  [680] = {x=34.462, y=0.000, z=-5.329, rx=-0.000, ry=0.000, rz=-0.000, shoulder=lefty, elbow=epositive, wrist=wpositive, fatherId=fReference[0]}
  [681] = {x=33.526, y=0.000, z=-5.347, rx=-0.000, ry=0.000, rz=-0.000, shoulder=lefty, elbow=epositive, wrist=wpositive, fatherId=fReference[0]}
  [682] = {x=32.941, y=0.000, z=-5.345, rx=-0.000, ry=0.000, rz=-0.000, shoulder=lefty, elbow=epositive, wrist=wpositive, fatherId=fReference[0]}
  [683] = {x=32.394, y=0.000, z=-5.347, rx=-0.000, ry=0.000, rz=-0.000, shoulder=lefty, elbow=epositive, wrist=wpositive, fatherId=fReference[0]}
  [684] = {x=31.868, y=0.000, z=-5.351, rx=-0.000, ry=0.000, rz=-0.000, shoulder=lefty, elbow=epositive, wrist=wpositive, fatherId=fReference[0]}
  [685] = {x=31.351, y=0.000, z=-5.356, rx=-0.000, ry=0.000, rz=-0.000, shoulder=lefty, elbow=epositive, wrist=wpositive, fatherId=fReference[0]}
  [686] = {x=30.840, y=0.000, z=-5.362, rx=-0.000, ry=0.000, rz=-0.000, shoulder=lefty, elbow=epositive, wrist=wpositive, fatherId=fReference[0]}
  [687] = {x=30.332, y=0.000, z=-5.369, rx=-0.000, ry=0.000, rz=-0.000, shoulder=lefty, elbow=epositive, wrist=wpositive, fatherId=fReference[0]}
  [688] = {x=29.826, y=0.000, z=-5.375, rx=-0.000, ry=0.000, rz=-0.000, shoulder=lefty, elbow=epositive, wrist=wpositive, fatherId=fReference[0]}
  [689] = {x=29.322, y=0.000, z=-5.383, rx=-0.000, ry=0.000, rz=-0.000, shoulder=lefty, elbow=epositive, wrist=wpositive, fatherId=fReference[0]}
  [690] = {x=28.818, y=0.000, z=-5.390, rx=-0.000, ry=0.000, rz=-0.000, shoulder=lefty, elbow=epositive, wrist=wpositive, fatherId=fReference[0]}
  [691] = {x=28.316, y=0.000, z=-5.397, rx=-0.000, ry=0.000, rz=-0.000, shoulder=lefty, elbow=epositive, wrist=wpositive, fatherId=fReference[0]}
  [692] = {x=27.814, y=0.000, z=-5.405, rx=-0.000, ry=0.000, rz=-0.000, shoulder=lefty, elbow=epositive, wrist=wpositive, fatherId=fReference[0]}
  [693] = {x=27.312, y=0.000, z=-5.413, rx=-0.000, ry=0.000, rz=-0.000, shoulder=lefty, elbow=epositive, wrist=wpositive, fatherId=fReference[0]}
  [694] = {x=26.812, y=0.000, z=-5.421, rx=-0.000, ry=0.000, rz=-0.000, shoulder=lefty, elbow=epositive, wrist=wpositive, fatherId=fReference[0]}
  [695] = {x=26.312, y=0.000, z=-5.429, rx=-0.000, ry=0.000, rz=-0.000, shoulder=lefty, elbow=epositive, wrist=wpositive, fatherId=fReference[0]}
  [696] = {x=25.812, y=0.000, z=-5.437, rx=-0.000, ry=0.000, rz=-0.000, shoulder=lefty, elbow=epositive, wrist=wpositive, fatherId=fReference[0]}
  [697] = {x=25.313, y=0.000, z=-5.446, rx=-0.000, ry=0.000, rz=-0.000, shoulder=lefty, elbow=epositive, wrist=wpositive, fatherId=fReference[0]}
  [698] = {x=24.813, y=0.000, z=-5.454, rx=-0.000, ry=0.000, rz=-0.000, shoulder=lefty, elbow=epositive, wrist=wpositive, fatherId=fReference[0]}
  [699] = {x=24.314, y=0.000, z=-5.462, rx=-0.000, ry=0.000, rz=-0.000, shoulder=lefty, elbow=epositive, wrist=wpositive, fatherId=fReference[0]}
  [700] = {x=23.815, y=0.000, z=-5.471, rx=-0.000, ry=0.000, rz=-0.000, shoulder=lefty, elbow=epositive, wrist=wpositive, fatherId=fReference[0]}
  [701] = {x=23.315, y=0.000, z=-5.479, rx=-0.000, ry=0.000, rz=-0.000, shoulder=lefty, elbow=epositive, wrist=wpositive, fatherId=fReference[0]}
  [702] = {x=22.816, y=0.000, z=-5.487, rx=-0.000, ry=0.000, rz=-0.000, shoulder=lefty, elbow=epositive, wrist=wpositive, fatherId=fReference[0]}
  [703] = {x=22.317, y=0.000, z=-5.496, rx=-0.000, ry=0.000, rz=-0.000, shoulder=lefty, elbow=epositive, wrist=wpositive, fatherId=fReference[0]}
  [704] = {x=21.818, y=0.000, z=-5.504, rx=-0.000, ry=0.000, rz=-0.000, shoulder=lefty, elbow=epositive, wrist=wpositive, fatherId=fReference[0]}
  [705] = {x=21.319, y=0.000, z=-5.513, rx=-0.000, ry=0.000, rz=-0.000, shoulder=lefty, elbow=epositive, wrist=wpositive, fatherId=fReference[0]}
  [706] = {x=20.820, y=0.000, z=-5.521, rx=-0.000, ry=0.000, rz=-0.000, shoulder=lefty, elbow=epositive, wrist=wpositive, fatherId=fReference[0]}
  [707] = {x=20.321, y=0.000, z=-5.530, rx=-0.000, ry=0.000, rz=-0.000, shoulder=lefty, elbow=epositive, wrist=wpositive, fatherId=fReference[0]}
  [708] = {x=19.823, y=0.000, z=-5.539, rx=-0.000, ry=0.000, rz=-0.000, shoulder=lefty, elbow=epositive, wrist=wpositive, fatherId=fReference[0]}
  [709] = {x=19.325, y=0.000, z=-5.548, rx=-0.000, ry=0.000, rz=-0.000, shoulder=lefty, elbow=epositive, wrist=wpositive, fatherId=fReference[0]}
  [710] = {x=18.827, y=0.000, z=-5.557, rx=-0.000, ry=0.000, rz=-0.000, shoulder=lefty, elbow=epositive, wrist=wpositive, fatherId=fReference[0]}
  [711] = {x=18.328, y=0.000, z=-5.565, rx=-0.000, ry=0.000, rz=-0.000, shoulder=lefty, elbow=epositive, wrist=wpositive, fatherId=fReference[0]}
  [712] = {x=17.830, y=0.000, z=-5.575, rx=-0.000, ry=0.000, rz=-0.000, shoulder=lefty, elbow=epositive, wrist=wpositive, fatherId=fReference[0]}
  [713] = {x=17.331, y=0.000, z=-5.583, rx=-0.000, ry=0.000, rz=-0.000, shoulder=lefty, elbow=epositive, wrist=wpositive, fatherId=fReference[0]}
  [714] = {x=16.833, y=0.000, z=-5.593, rx=-0.000, ry=0.000, rz=-0.000, shoulder=lefty, elbow=epositive, wrist=wpositive, fatherId=fReference[0]}
  [715] = {x=16.335, y=0.000, z=-5.601, rx=-0.000, ry=0.000, rz=-0.000, shoulder=lefty, elbow=epositive, wrist=wpositive, fatherId=fReference[0]}
  [716] = {x=15.836, y=0.000, z=-5.611, rx=-0.000, ry=0.000, rz=-0.000, shoulder=lefty, elbow=epositive, wrist=wpositive, fatherId=fReference[0]}
  [717] = {x=15.338, y=0.000, z=-5.620, rx=-0.000, ry=0.000, rz=-0.000, shoulder=lefty, elbow=epositive, wrist=wpositive, fatherId=fReference[0]}
  [718] = {x=14.840, y=0.000, z=-5.628, rx=-0.000, ry=0.000, rz=-0.000, shoulder=lefty, elbow=epositive, wrist=wpositive, fatherId=fReference[0]}
  [719] = {x=14.342, y=0.000, z=-5.638, rx=-0.000, ry=0.000, rz=-0.000, shoulder=lefty, elbow=epositive, wrist=wpositive, fatherId=fReference[0]}
  [720] = {x=13.843, y=0.000, z=-5.646, rx=-0.000, ry=0.000, rz=-0.000, shoulder=lefty, elbow=epositive, wrist=wpositive, fatherId=fReference[0]}
  [721] = {x=13.344, y=0.000, z=-5.655, rx=-0.000, ry=0.000, rz=-0.000, shoulder=lefty, elbow=epositive, wrist=wpositive, fatherId=fReference[0]}
  [722] = {x=12.846, y=0.000, z=-5.664, rx=-0.000, ry=0.000, rz=-0.000, shoulder=lefty, elbow=epositive, wrist=wpositive, fatherId=fReference[0]}
  [723] = {x=12.345, y=0.000, z=-5.673, rx=-0.000, ry=0.000, rz=-0.000, shoulder=lefty, elbow=epositive, wrist=wpositive, fatherId=fReference[0]}
  [724] = {x=11.846, y=0.000, z=-5.682, rx=-0.000, ry=0.000, rz=-0.000, shoulder=lefty, elbow=epositive, wrist=wpositive, fatherId=fReference[0]}
  [725] = {x=11.347, y=0.000, z=-5.690, rx=-0.000, ry=0.000, rz=-0.000, shoulder=lefty, elbow=epositive, wrist=wpositive, fatherId=fReference[0]}
  [726] = {x=10.847, y=0.000, z=-5.699, rx=-0.000, ry=0.000, rz=-0.000, shoulder=lefty, elbow=epositive, wrist=wpositive, fatherId=fReference[0]}
  [727] = {x=10.347, y=0.000, z=-5.707, rx=-0.000, ry=0.000, rz=-0.000, shoulder=lefty, elbow=epositive, wrist=wpositive, fatherId=fReference[0]}
  [728] = {x=9.846, y=0.000, z=-5.716, rx=-0.000, ry=0.000, rz=-0.000, shoulder=lefty, elbow=epositive, wrist=wpositive, fatherId=fReference[0]}
  [729] = {x=9.346, y=0.000, z=-5.724, rx=-0.000, ry=0.000, rz=-0.000, shoulder=lefty, elbow=epositive, wrist=wpositive, fatherId=fReference[0]}
  [730] = {x=8.847, y=0.000, z=-5.733, rx=-0.000, ry=0.000, rz=-0.000, shoulder=lefty, elbow=epositive, wrist=wpositive, fatherId=fReference[0]}
  [731] = {x=8.346, y=0.000, z=-5.741, rx=-0.000, ry=0.000, rz=-0.000, shoulder=lefty, elbow=epositive, wrist=wpositive, fatherId=fReference[0]}
  [732] = {x=7.846, y=0.000, z=-5.750, rx=-0.000, ry=0.000, rz=-0.000, shoulder=lefty, elbow=epositive, wrist=wpositive, fatherId=fReference[0]}
  [733] = {x=7.344, y=0.000, z=-5.758, rx=-0.000, ry=0.000, rz=-0.000, shoulder=lefty, elbow=epositive, wrist=wpositive, fatherId=fReference[0]}
  [734] = {x=6.843, y=0.000, z=-5.766, rx=-0.000, ry=0.000, rz=-0.000, shoulder=lefty, elbow=epositive, wrist=wpositive, fatherId=fReference[0]}
  [735] = {x=6.341, y=0.000, z=-5.774, rx=-0.000, ry=0.000, rz=-0.000, shoulder=lefty, elbow=epositive, wrist=wpositive, fatherId=fReference[0]}
  [736] = {x=5.838, y=0.000, z=-5.782, rx=-0.000, ry=0.000, rz=-0.000, shoulder=lefty, elbow=epositive, wrist=wpositive, fatherId=fReference[0]}
  [737] = {x=5.336, y=0.000, z=-5.791, rx=-0.000, ry=0.000, rz=-0.000, shoulder=lefty, elbow=epositive, wrist=wpositive, fatherId=fReference[0]}
  [738] = {x=4.831, y=0.000, z=-5.798, rx=-0.000, ry=0.000, rz=-0.000, shoulder=lefty, elbow=epositive, wrist=wpositive, fatherId=fReference[0]}
  [739] = {x=4.326, y=0.000, z=-5.806, rx=-0.000, ry=0.000, rz=-0.000, shoulder=lefty, elbow=epositive, wrist=wpositive, fatherId=fReference[0]}
  [740] = {x=3.823, y=0.000, z=-5.814, rx=-0.000, ry=0.000, rz=-0.000, shoulder=lefty, elbow=epositive, wrist=wpositive, fatherId=fReference[0]}
  [741] = {x=3.321, y=0.000, z=-5.822, rx=-0.000, ry=0.000, rz=-0.000, shoulder=lefty, elbow=epositive, wrist=wpositive, fatherId=fReference[0]}
  [742] = {x=2.818, y=0.000, z=-5.830, rx=-0.000, ry=0.000, rz=-0.000, shoulder=lefty, elbow=epositive, wrist=wpositive, fatherId=fReference[0]}
  [743] = {x=2.316, y=0.000, z=-5.838, rx=-0.000, ry=0.000, rz=-0.000, shoulder=lefty, elbow=epositive, wrist=wpositive, fatherId=fReference[0]}
  [744] = {x=1.816, y=0.000, z=-5.847, rx=-0.000, ry=0.000, rz=-0.000, shoulder=lefty, elbow=epositive, wrist=wpositive, fatherId=fReference[0]}
  [745] = {x=1.313, y=0.000, z=-5.855, rx=-0.000, ry=0.000, rz=-0.000, shoulder=lefty, elbow=epositive, wrist=wpositive, fatherId=fReference[0]}
  [746] = {x=0.814, y=0.000, z=-5.864, rx=-0.000, ry=0.000, rz=-0.000, shoulder=lefty, elbow=epositive, wrist=wpositive, fatherId=fReference[0]}
  [747] = {x=0.312, y=0.000, z=-5.872, rx=-0.000, ry=0.000, rz=-0.000, shoulder=lefty, elbow=epositive, wrist=wpositive, fatherId=fReference[0]}
  [748] = {x=-0.190, y=0.000, z=-5.880, rx=-0.000, ry=0.000, rz=-0.000, shoulder=lefty, elbow=epositive, wrist=wpositive, fatherId=fReference[0]}
  [749] = {x=-0.691, y=0.000, z=-5.889, rx=-0.000, ry=0.000, rz=-0.000, shoulder=lefty, elbow=epositive, wrist=wpositive, fatherId=fReference[0]}
  [750] = {x=-1.192, y=0.000, z=-5.897, rx=-0.000, ry=0.000, rz=-0.000, shoulder=lefty, elbow=epositive, wrist=wpositive, fatherId=fReference[0]}
  [751] = {x=-1.693, y=0.000, z=-5.906, rx=-0.000, ry=0.000, rz=-0.000, shoulder=lefty, elbow=epositive, wrist=wpositive, fatherId=fReference[0]}
  [752] = {x=-2.194, y=0.000, z=-5.915, rx=-0.000, ry=0.000, rz=-0.000, shoulder=lefty, elbow=epositive, wrist=wpositive, fatherId=fReference[0]}
  [753] = {x=-2.695, y=0.000, z=-5.923, rx=-0.000, ry=0.000, rz=-0.000, shoulder=lefty, elbow=epositive, wrist=wpositive, fatherId=fReference[0]}
  [754] = {x=-3.197, y=0.000, z=-5.932, rx=-0.000, ry=0.000, rz=-0.000, shoulder=lefty, elbow=epositive, wrist=wpositive, fatherId=fReference[0]}
  [755] = {x=-3.697, y=0.000, z=-5.941, rx=-0.000, ry=0.000, rz=-0.000, shoulder=lefty, elbow=epositive, wrist=wpositive, fatherId=fReference[0]}
  [756] = {x=-4.197, y=0.000, z=-5.950, rx=-0.000, ry=0.000, rz=-0.000, shoulder=lefty, elbow=epositive, wrist=wpositive, fatherId=fReference[0]}
  [757] = {x=-4.697, y=0.000, z=-5.959, rx=-0.000, ry=0.000, rz=-0.000, shoulder=lefty, elbow=epositive, wrist=wpositive, fatherId=fReference[0]}
  [758] = {x=-5.197, y=0.000, z=-5.968, rx=-0.000, ry=0.000, rz=-0.000, shoulder=lefty, elbow=epositive, wrist=wpositive, fatherId=fReference[0]}
  [759] = {x=-5.696, y=0.000, z=-5.977, rx=-0.000, ry=0.000, rz=-0.000, shoulder=lefty, elbow=epositive, wrist=wpositive, fatherId=fReference[0]}
  [760] = {x=-6.198, y=0.000, z=-5.985, rx=-0.000, ry=0.000, rz=-0.000, shoulder=lefty, elbow=epositive, wrist=wpositive, fatherId=fReference[0]}
  [761] = {x=-6.700, y=0.000, z=-5.994, rx=-0.000, ry=0.000, rz=-0.000, shoulder=lefty, elbow=epositive, wrist=wpositive, fatherId=fReference[0]}
  [762] = {x=-7.198, y=0.000, z=-6.004, rx=-0.000, ry=0.000, rz=-0.000, shoulder=lefty, elbow=epositive, wrist=wpositive, fatherId=fReference[0]}
  [763] = {x=-7.696, y=0.000, z=-6.013, rx=-0.000, ry=0.000, rz=-0.000, shoulder=lefty, elbow=epositive, wrist=wpositive, fatherId=fReference[0]}
  [764] = {x=-8.197, y=0.000, z=-6.022, rx=-0.000, ry=0.000, rz=-0.000, shoulder=lefty, elbow=epositive, wrist=wpositive, fatherId=fReference[0]}
  [765] = {x=-8.698, y=0.000, z=-6.031, rx=-0.000, ry=0.000, rz=-0.000, shoulder=lefty, elbow=epositive, wrist=wpositive, fatherId=fReference[0]}
  [766] = {x=-9.196, y=0.000, z=-6.040, rx=-0.000, ry=0.000, rz=-0.000, shoulder=lefty, elbow=epositive, wrist=wpositive, fatherId=fReference[0]}
  [767] = {x=-9.696, y=0.000, z=-6.050, rx=-0.000, ry=0.000, rz=-0.000, shoulder=lefty, elbow=epositive, wrist=wpositive, fatherId=fReference[0]}
  [768] = {x=-10.193, y=0.000, z=-6.060, rx=-0.000, ry=0.000, rz=-0.000, shoulder=lefty, elbow=epositive, wrist=wpositive, fatherId=fReference[0]}
  [769] = {x=-10.692, y=0.000, z=-6.069, rx=-0.000, ry=0.000, rz=-0.000, shoulder=lefty, elbow=epositive, wrist=wpositive, fatherId=fReference[0]}
  [770] = {x=-11.189, y=0.000, z=-6.079, rx=-0.000, ry=0.000, rz=-0.000, shoulder=lefty, elbow=epositive, wrist=wpositive, fatherId=fReference[0]}
  [771] = {x=-11.687, y=0.000, z=-6.088, rx=-0.000, ry=0.000, rz=-0.000, shoulder=lefty, elbow=epositive, wrist=wpositive, fatherId=fReference[0]}
  [772] = {x=-12.183, y=0.000, z=-6.098, rx=-0.000, ry=0.000, rz=-0.000, shoulder=lefty, elbow=epositive, wrist=wpositive, fatherId=fReference[0]}
  [773] = {x=-12.685, y=0.000, z=-6.108, rx=-0.000, ry=0.000, rz=-0.000, shoulder=lefty, elbow=epositive, wrist=wpositive, fatherId=fReference[0]}
  [774] = {x=-13.181, y=0.000, z=-6.117, rx=-0.000, ry=0.000, rz=-0.000, shoulder=lefty, elbow=epositive, wrist=wpositive, fatherId=fReference[0]}
  [775] = {x=-13.678, y=0.000, z=-6.127, rx=-0.000, ry=0.000, rz=-0.000, shoulder=lefty, elbow=epositive, wrist=wpositive, fatherId=fReference[0]}
  [776] = {x=-14.176, y=0.000, z=-6.137, rx=-0.000, ry=0.000, rz=-0.000, shoulder=lefty, elbow=epositive, wrist=wpositive, fatherId=fReference[0]}
  [777] = {x=-14.670, y=0.000, z=-6.147, rx=-0.000, ry=0.000, rz=-0.000, shoulder=lefty, elbow=epositive, wrist=wpositive, fatherId=fReference[0]}
  [778] = {x=-15.170, y=0.000, z=-6.157, rx=-0.000, ry=0.000, rz=-0.000, shoulder=lefty, elbow=epositive, wrist=wpositive, fatherId=fReference[0]}
  [779] = {x=-15.665, y=0.000, z=-6.167, rx=-0.000, ry=0.000, rz=-0.000, shoulder=lefty, elbow=epositive, wrist=wpositive, fatherId=fReference[0]}
  [780] = {x=-16.162, y=0.000, z=-6.177, rx=-0.000, ry=0.000, rz=-0.000, shoulder=lefty, elbow=epositive, wrist=wpositive, fatherId=fReference[0]}
  [781] = {x=-16.658, y=0.000, z=-6.188, rx=-0.000, ry=0.000, rz=-0.000, shoulder=lefty, elbow=epositive, wrist=wpositive, fatherId=fReference[0]}
  [782] = {x=-17.157, y=0.000, z=-6.197, rx=-0.000, ry=0.000, rz=-0.000, shoulder=lefty, elbow=epositive, wrist=wpositive, fatherId=fReference[0]}
  [783] = {x=-17.653, y=0.000, z=-6.207, rx=-0.000, ry=0.000, rz=-0.000, shoulder=lefty, elbow=epositive, wrist=wpositive, fatherId=fReference[0]}
  [784] = {x=-18.149, y=0.000, z=-6.218, rx=-0.000, ry=0.000, rz=-0.000, shoulder=lefty, elbow=epositive, wrist=wpositive, fatherId=fReference[0]}
  [785] = {x=-18.646, y=0.000, z=-6.228, rx=-0.000, ry=0.000, rz=-0.000, shoulder=lefty, elbow=epositive, wrist=wpositive, fatherId=fReference[0]}
  [786] = {x=-19.137, y=0.000, z=-6.239, rx=-0.000, ry=0.000, rz=-0.000, shoulder=lefty, elbow=epositive, wrist=wpositive, fatherId=fReference[0]}
  [787] = {x=-19.637, y=0.000, z=-6.248, rx=-0.000, ry=0.000, rz=-0.000, shoulder=lefty, elbow=epositive, wrist=wpositive, fatherId=fReference[0]}
  [788] = {x=-20.133, y=0.000, z=-6.259, rx=-0.000, ry=0.000, rz=-0.000, shoulder=lefty, elbow=epositive, wrist=wpositive, fatherId=fReference[0]}
  [789] = {x=-20.628, y=0.000, z=-6.269, rx=-0.000, ry=0.000, rz=-0.000, shoulder=lefty, elbow=epositive, wrist=wpositive, fatherId=fReference[0]}
  [790] = {x=-21.125, y=0.000, z=-6.279, rx=-0.000, ry=0.000, rz=-0.000, shoulder=lefty, elbow=epositive, wrist=wpositive, fatherId=fReference[0]}
  [791] = {x=-21.624, y=0.000, z=-6.289, rx=-0.000, ry=0.000, rz=-0.000, shoulder=lefty, elbow=epositive, wrist=wpositive, fatherId=fReference[0]}
  [792] = {x=-22.120, y=0.000, z=-6.300, rx=-0.000, ry=0.000, rz=-0.000, shoulder=lefty, elbow=epositive, wrist=wpositive, fatherId=fReference[0]}
  [793] = {x=-22.612, y=0.000, z=-6.311, rx=-0.000, ry=0.000, rz=-0.000, shoulder=lefty, elbow=epositive, wrist=wpositive, fatherId=fReference[0]}
  [794] = {x=-23.110, y=0.000, z=-6.322, rx=-0.000, ry=0.000, rz=-0.000, shoulder=lefty, elbow=epositive, wrist=wpositive, fatherId=fReference[0]}
  [795] = {x=-23.609, y=0.000, z=-6.332, rx=-0.000, ry=0.000, rz=-0.000, shoulder=lefty, elbow=epositive, wrist=wpositive, fatherId=fReference[0]}
  [796] = {x=-24.107, y=0.000, z=-6.343, rx=-0.000, ry=0.000, rz=-0.000, shoulder=lefty, elbow=epositive, wrist=wpositive, fatherId=fReference[0]}
  [797] = {x=-24.603, y=0.000, z=-6.354, rx=-0.000, ry=0.000, rz=-0.000, shoulder=lefty, elbow=epositive, wrist=wpositive, fatherId=fReference[0]}
  [798] = {x=-25.098, y=0.000, z=-6.365, rx=-0.000, ry=0.000, rz=-0.000, shoulder=lefty, elbow=epositive, wrist=wpositive, fatherId=fReference[0]}
  [799] = {x=-25.593, y=0.000, z=-6.377, rx=-0.000, ry=0.000, rz=-0.000, shoulder=lefty, elbow=epositive, wrist=wpositive, fatherId=fReference[0]}
  [800] = {x=-26.088, y=0.000, z=-6.388, rx=-0.000, ry=0.000, rz=-0.000, shoulder=lefty, elbow=epositive, wrist=wpositive, fatherId=fReference[0]}
  [801] = {x=-26.584, y=0.000, z=-6.400, rx=-0.000, ry=0.000, rz=-0.000, shoulder=lefty, elbow=epositive, wrist=wpositive, fatherId=fReference[0]}
  [802] = {x=-27.083, y=0.000, z=-6.412, rx=-0.000, ry=0.000, rz=-0.000, shoulder=lefty, elbow=epositive, wrist=wpositive, fatherId=fReference[0]}
  [803] = {x=-27.583, y=0.000, z=-6.423, rx=-0.000, ry=0.000, rz=-0.000, shoulder=lefty, elbow=epositive, wrist=wpositive, fatherId=fReference[0]}
  [804] = {x=-28.088, y=0.000, z=-6.434, rx=-0.000, ry=0.000, rz=-0.000, shoulder=lefty, elbow=epositive, wrist=wpositive, fatherId=fReference[0]}
  [805] = {x=-28.594, y=0.000, z=-6.445, rx=-0.000, ry=0.000, rz=-0.000, shoulder=lefty, elbow=epositive, wrist=wpositive, fatherId=fReference[0]}
  [806] = {x=-29.107, y=0.000, z=-6.455, rx=-0.000, ry=0.000, rz=-0.000, shoulder=lefty, elbow=epositive, wrist=wpositive, fatherId=fReference[0]}
  [807] = {x=-29.626, y=0.000, z=-6.466, rx=-0.000, ry=0.000, rz=-0.000, shoulder=lefty, elbow=epositive, wrist=wpositive, fatherId=fReference[0]}
  [808] = {x=-30.142, y=0.000, z=-6.476, rx=-0.000, ry=0.000, rz=-0.000, shoulder=lefty, elbow=epositive, wrist=wpositive, fatherId=fReference[0]}
  [809] = {x=-30.665, y=0.000, z=-6.487, rx=-0.000, ry=0.000, rz=-0.000, shoulder=lefty, elbow=epositive, wrist=wpositive, fatherId=fReference[0]}
  [810] = {x=-31.185, y=0.000, z=-6.496, rx=-0.000, ry=0.000, rz=-0.000, shoulder=lefty, elbow=epositive, wrist=wpositive, fatherId=fReference[0]}
  [811] = {x=-30.257, y=0.000, z=-6.431, rx=-0.000, ry=0.000, rz=-0.000, shoulder=lefty, elbow=epositive, wrist=wpositive, fatherId=fReference[0]}
  [812] = {x=-29.750, y=0.000, z=-6.417, rx=-0.000, ry=0.000, rz=-0.000, shoulder=lefty, elbow=epositive, wrist=wpositive, fatherId=fReference[0]}
  [813] = {x=-29.239, y=0.000, z=-6.413, rx=-0.000, ry=0.000, rz=-0.000, shoulder=lefty, elbow=epositive, wrist=wpositive, fatherId=fReference[0]}
  [814] = {x=-28.740, y=0.000, z=-6.414, rx=-0.000, ry=0.000, rz=-0.000, shoulder=lefty, elbow=epositive, wrist=wpositive, fatherId=fReference[0]}
  [815] = {x=-28.245, y=0.000, z=-6.417, rx=-0.000, ry=0.000, rz=-0.000, shoulder=lefty, elbow=epositive, wrist=wpositive, fatherId=fReference[0]}
  [816] = {x=-27.750, y=0.000, z=-6.422, rx=-0.000, ry=0.000, rz=-0.000, shoulder=lefty, elbow=epositive, wrist=wpositive, fatherId=fReference[0]}
  [817] = {x=-27.253, y=0.000, z=-6.428, rx=-0.000, ry=0.000, rz=-0.000, shoulder=lefty, elbow=epositive, wrist=wpositive, fatherId=fReference[0]}
  [818] = {x=-26.756, y=0.000, z=-6.434, rx=-0.000, ry=0.000, rz=-0.000, shoulder=lefty, elbow=epositive, wrist=wpositive, fatherId=fReference[0]}
  [819] = {x=-26.258, y=0.000, z=-6.440, rx=-0.000, ry=0.000, rz=-0.000, shoulder=lefty, elbow=epositive, wrist=wpositive, fatherId=fReference[0]}
  [820] = {x=-25.760, y=0.000, z=-6.447, rx=-0.000, ry=0.000, rz=-0.000, shoulder=lefty, elbow=epositive, wrist=wpositive, fatherId=fReference[0]}
  [821] = {x=-25.260, y=0.000, z=-6.454, rx=-0.000, ry=0.000, rz=-0.000, shoulder=lefty, elbow=epositive, wrist=wpositive, fatherId=fReference[0]}
  [822] = {x=-24.760, y=0.000, z=-6.461, rx=-0.000, ry=0.000, rz=-0.000, shoulder=lefty, elbow=epositive, wrist=wpositive, fatherId=fReference[0]}
  [823] = {x=-24.258, y=0.000, z=-6.468, rx=-0.000, ry=0.000, rz=-0.000, shoulder=lefty, elbow=epositive, wrist=wpositive, fatherId=fReference[0]}
  [824] = {x=-23.754, y=0.000, z=-6.476, rx=-0.000, ry=0.000, rz=-0.000, shoulder=lefty, elbow=epositive, wrist=wpositive, fatherId=fReference[0]}
  [825] = {x=-23.252, y=0.000, z=-6.484, rx=-0.000, ry=0.000, rz=-0.000, shoulder=lefty, elbow=epositive, wrist=wpositive, fatherId=fReference[0]}
  [826] = {x=-22.750, y=0.000, z=-6.493, rx=-0.000, ry=0.000, rz=-0.000, shoulder=lefty, elbow=epositive, wrist=wpositive, fatherId=fReference[0]}
  [827] = {x=-22.246, y=0.000, z=-6.501, rx=-0.000, ry=0.000, rz=-0.000, shoulder=lefty, elbow=epositive, wrist=wpositive, fatherId=fReference[0]}
  [828] = {x=-21.743, y=0.000, z=-6.509, rx=-0.000, ry=0.000, rz=-0.000, shoulder=lefty, elbow=epositive, wrist=wpositive, fatherId=fReference[0]}
  [829] = {x=-21.239, y=0.000, z=-6.517, rx=-0.000, ry=0.000, rz=-0.000, shoulder=lefty, elbow=epositive, wrist=wpositive, fatherId=fReference[0]}
  [830] = {x=-20.736, y=0.000, z=-6.526, rx=-0.000, ry=0.000, rz=-0.000, shoulder=lefty, elbow=epositive, wrist=wpositive, fatherId=fReference[0]}
  [831] = {x=-20.232, y=0.000, z=-6.534, rx=-0.000, ry=0.000, rz=-0.000, shoulder=lefty, elbow=epositive, wrist=wpositive, fatherId=fReference[0]}
  [832] = {x=-19.728, y=0.000, z=-6.542, rx=-0.000, ry=0.000, rz=-0.000, shoulder=lefty, elbow=epositive, wrist=wpositive, fatherId=fReference[0]}
  [833] = {x=-19.225, y=0.000, z=-6.551, rx=-0.000, ry=0.000, rz=-0.000, shoulder=lefty, elbow=epositive, wrist=wpositive, fatherId=fReference[0]}
  [834] = {x=-18.722, y=0.000, z=-6.559, rx=-0.000, ry=0.000, rz=-0.000, shoulder=lefty, elbow=epositive, wrist=wpositive, fatherId=fReference[0]}
  [835] = {x=-18.218, y=0.000, z=-6.567, rx=-0.000, ry=0.000, rz=-0.000, shoulder=lefty, elbow=epositive, wrist=wpositive, fatherId=fReference[0]}
  [836] = {x=-17.714, y=0.000, z=-6.575, rx=-0.000, ry=0.000, rz=-0.000, shoulder=lefty, elbow=epositive, wrist=wpositive, fatherId=fReference[0]}
  [837] = {x=-17.210, y=0.000, z=-6.583, rx=-0.000, ry=0.000, rz=-0.000, shoulder=lefty, elbow=epositive, wrist=wpositive, fatherId=fReference[0]}
  [838] = {x=-16.706, y=0.000, z=-6.591, rx=-0.000, ry=0.000, rz=-0.000, shoulder=lefty, elbow=epositive, wrist=wpositive, fatherId=fReference[0]}
  [839] = {x=-16.203, y=0.000, z=-6.599, rx=-0.000, ry=0.000, rz=-0.000, shoulder=lefty, elbow=epositive, wrist=wpositive, fatherId=fReference[0]}
  [840] = {x=-15.699, y=0.000, z=-6.608, rx=-0.000, ry=0.000, rz=-0.000, shoulder=lefty, elbow=epositive, wrist=wpositive, fatherId=fReference[0]}
  [841] = {x=-15.195, y=0.000, z=-6.616, rx=-0.000, ry=0.000, rz=-0.000, shoulder=lefty, elbow=epositive, wrist=wpositive, fatherId=fReference[0]}
  [842] = {x=-14.690, y=0.000, z=-6.624, rx=-0.000, ry=0.000, rz=-0.000, shoulder=lefty, elbow=epositive, wrist=wpositive, fatherId=fReference[0]}
  [843] = {x=-14.187, y=0.000, z=-6.632, rx=-0.000, ry=0.000, rz=-0.000, shoulder=lefty, elbow=epositive, wrist=wpositive, fatherId=fReference[0]}
  [844] = {x=-13.683, y=0.000, z=-6.641, rx=-0.000, ry=0.000, rz=-0.000, shoulder=lefty, elbow=epositive, wrist=wpositive, fatherId=fReference[0]}
  [845] = {x=-13.177, y=0.000, z=-6.649, rx=-0.000, ry=0.000, rz=-0.000, shoulder=lefty, elbow=epositive, wrist=wpositive, fatherId=fReference[0]}
  [846] = {x=-12.673, y=0.000, z=-6.657, rx=-0.000, ry=0.000, rz=-0.000, shoulder=lefty, elbow=epositive, wrist=wpositive, fatherId=fReference[0]}
  [847] = {x=-12.168, y=0.000, z=-6.665, rx=-0.000, ry=0.000, rz=-0.000, shoulder=lefty, elbow=epositive, wrist=wpositive, fatherId=fReference[0]}
  [848] = {x=-11.664, y=0.000, z=-6.674, rx=-0.000, ry=0.000, rz=-0.000, shoulder=lefty, elbow=epositive, wrist=wpositive, fatherId=fReference[0]}
  [849] = {x=-11.159, y=0.000, z=-6.682, rx=-0.000, ry=0.000, rz=-0.000, shoulder=lefty, elbow=epositive, wrist=wpositive, fatherId=fReference[0]}
  [850] = {x=-10.654, y=0.000, z=-6.691, rx=-0.000, ry=0.000, rz=-0.000, shoulder=lefty, elbow=epositive, wrist=wpositive, fatherId=fReference[0]}
  [851] = {x=-10.149, y=0.000, z=-6.699, rx=-0.000, ry=0.000, rz=-0.000, shoulder=lefty, elbow=epositive, wrist=wpositive, fatherId=fReference[0]}
  [852] = {x=-9.643, y=0.000, z=-6.708, rx=-0.000, ry=0.000, rz=-0.000, shoulder=lefty, elbow=epositive, wrist=wpositive, fatherId=fReference[0]}
  [853] = {x=-9.136, y=0.000, z=-6.717, rx=-0.000, ry=0.000, rz=-0.000, shoulder=lefty, elbow=epositive, wrist=wpositive, fatherId=fReference[0]}
  [854] = {x=-8.629, y=0.000, z=-6.725, rx=-0.000, ry=0.000, rz=-0.000, shoulder=lefty, elbow=epositive, wrist=wpositive, fatherId=fReference[0]}
  [855] = {x=-8.124, y=0.000, z=-6.734, rx=-0.000, ry=0.000, rz=-0.000, shoulder=lefty, elbow=epositive, wrist=wpositive, fatherId=fReference[0]}
  [856] = {x=-7.618, y=0.000, z=-6.743, rx=-0.000, ry=0.000, rz=-0.000, shoulder=lefty, elbow=epositive, wrist=wpositive, fatherId=fReference[0]}
  [857] = {x=-7.111, y=0.000, z=-6.752, rx=-0.000, ry=0.000, rz=-0.000, shoulder=lefty, elbow=epositive, wrist=wpositive, fatherId=fReference[0]}
  [858] = {x=-6.605, y=0.000, z=-6.759, rx=-0.000, ry=0.000, rz=-0.000, shoulder=lefty, elbow=epositive, wrist=wpositive, fatherId=fReference[0]}
  [859] = {x=-6.098, y=0.000, z=-6.768, rx=-0.000, ry=0.000, rz=-0.000, shoulder=lefty, elbow=epositive, wrist=wpositive, fatherId=fReference[0]}
  [860] = {x=-5.593, y=0.000, z=-6.776, rx=-0.000, ry=0.000, rz=-0.000, shoulder=lefty, elbow=epositive, wrist=wpositive, fatherId=fReference[0]}
  [861] = {x=-5.088, y=0.000, z=-6.784, rx=-0.000, ry=0.000, rz=-0.000, shoulder=lefty, elbow=epositive, wrist=wpositive, fatherId=fReference[0]}
  [862] = {x=-4.583, y=0.000, z=-6.792, rx=-0.000, ry=0.000, rz=-0.000, shoulder=lefty, elbow=epositive, wrist=wpositive, fatherId=fReference[0]}
  [863] = {x=-4.079, y=0.000, z=-6.799, rx=-0.000, ry=0.000, rz=-0.000, shoulder=lefty, elbow=epositive, wrist=wpositive, fatherId=fReference[0]}
  [864] = {x=-3.574, y=0.000, z=-6.807, rx=-0.000, ry=0.000, rz=-0.000, shoulder=lefty, elbow=epositive, wrist=wpositive, fatherId=fReference[0]}
  [865] = {x=-3.070, y=0.000, z=-6.815, rx=-0.000, ry=0.000, rz=-0.000, shoulder=lefty, elbow=epositive, wrist=wpositive, fatherId=fReference[0]}
  [866] = {x=-2.566, y=0.000, z=-6.821, rx=-0.000, ry=0.000, rz=-0.000, shoulder=lefty, elbow=epositive, wrist=wpositive, fatherId=fReference[0]}
  [867] = {x=-2.061, y=0.000, z=-6.830, rx=-0.000, ry=0.000, rz=-0.000, shoulder=lefty, elbow=epositive, wrist=wpositive, fatherId=fReference[0]}
  [868] = {x=-1.556, y=0.000, z=-6.838, rx=-0.000, ry=0.000, rz=-0.000, shoulder=lefty, elbow=epositive, wrist=wpositive, fatherId=fReference[0]}
  [869] = {x=-1.051, y=0.000, z=-6.845, rx=-0.000, ry=0.000, rz=-0.000, shoulder=lefty, elbow=epositive, wrist=wpositive, fatherId=fReference[0]}
  [870] = {x=-0.546, y=0.000, z=-6.854, rx=-0.000, ry=0.000, rz=-0.000, shoulder=lefty, elbow=epositive, wrist=wpositive, fatherId=fReference[0]}
  [871] = {x=-0.041, y=0.000, z=-6.861, rx=-0.000, ry=0.000, rz=-0.000, shoulder=lefty, elbow=epositive, wrist=wpositive, fatherId=fReference[0]}
  [872] = {x=0.465, y=0.000, z=-6.868, rx=-0.000, ry=0.000, rz=-0.000, shoulder=lefty, elbow=epositive, wrist=wpositive, fatherId=fReference[0]}
  [873] = {x=0.970, y=0.000, z=-6.877, rx=-0.000, ry=0.000, rz=-0.000, shoulder=lefty, elbow=epositive, wrist=wpositive, fatherId=fReference[0]}
  [874] = {x=1.475, y=0.000, z=-6.884, rx=-0.000, ry=0.000, rz=-0.000, shoulder=lefty, elbow=epositive, wrist=wpositive, fatherId=fReference[0]}
  [875] = {x=1.982, y=0.000, z=-6.892, rx=-0.000, ry=0.000, rz=-0.000, shoulder=lefty, elbow=epositive, wrist=wpositive, fatherId=fReference[0]}
  [876] = {x=2.487, y=0.000, z=-6.900, rx=-0.000, ry=0.000, rz=-0.000, shoulder=lefty, elbow=epositive, wrist=wpositive, fatherId=fReference[0]}
  [877] = {x=2.993, y=0.000, z=-6.908, rx=-0.000, ry=0.000, rz=-0.000, shoulder=lefty, elbow=epositive, wrist=wpositive, fatherId=fReference[0]}
  [878] = {x=3.500, y=0.000, z=-6.916, rx=-0.000, ry=0.000, rz=-0.000, shoulder=lefty, elbow=epositive, wrist=wpositive, fatherId=fReference[0]}
  [879] = {x=4.007, y=0.000, z=-6.925, rx=-0.000, ry=0.000, rz=-0.000, shoulder=lefty, elbow=epositive, wrist=wpositive, fatherId=fReference[0]}
  [880] = {x=4.514, y=0.000, z=-6.933, rx=-0.000, ry=0.000, rz=-0.000, shoulder=lefty, elbow=epositive, wrist=wpositive, fatherId=fReference[0]}
  [881] = {x=5.020, y=0.000, z=-6.941, rx=-0.000, ry=0.000, rz=-0.000, shoulder=lefty, elbow=epositive, wrist=wpositive, fatherId=fReference[0]}
  [882] = {x=5.528, y=0.000, z=-6.950, rx=-0.000, ry=0.000, rz=-0.000, shoulder=lefty, elbow=epositive, wrist=wpositive, fatherId=fReference[0]}
  [883] = {x=6.034, y=0.000, z=-6.958, rx=-0.000, ry=0.000, rz=-0.000, shoulder=lefty, elbow=epositive, wrist=wpositive, fatherId=fReference[0]}
  [884] = {x=6.541, y=0.000, z=-6.966, rx=-0.000, ry=0.000, rz=-0.000, shoulder=lefty, elbow=epositive, wrist=wpositive, fatherId=fReference[0]}
  [885] = {x=7.048, y=0.000, z=-6.975, rx=-0.000, ry=0.000, rz=-0.000, shoulder=lefty, elbow=epositive, wrist=wpositive, fatherId=fReference[0]}
  [886] = {x=7.555, y=0.000, z=-6.983, rx=-0.000, ry=0.000, rz=-0.000, shoulder=lefty, elbow=epositive, wrist=wpositive, fatherId=fReference[0]}
  [887] = {x=8.062, y=0.000, z=-6.992, rx=-0.000, ry=0.000, rz=-0.000, shoulder=lefty, elbow=epositive, wrist=wpositive, fatherId=fReference[0]}
  [888] = {x=8.568, y=0.000, z=-7.001, rx=-0.000, ry=0.000, rz=-0.000, shoulder=lefty, elbow=epositive, wrist=wpositive, fatherId=fReference[0]}
  [889] = {x=9.076, y=0.000, z=-7.010, rx=-0.000, ry=0.000, rz=-0.000, shoulder=lefty, elbow=epositive, wrist=wpositive, fatherId=fReference[0]}
  [890] = {x=9.586, y=0.000, z=-7.019, rx=-0.000, ry=0.000, rz=-0.000, shoulder=lefty, elbow=epositive, wrist=wpositive, fatherId=fReference[0]}
  [891] = {x=10.093, y=0.000, z=-7.028, rx=-0.000, ry=0.000, rz=-0.000, shoulder=lefty, elbow=epositive, wrist=wpositive, fatherId=fReference[0]}
  [892] = {x=10.601, y=0.000, z=-7.037, rx=-0.000, ry=0.000, rz=-0.000, shoulder=lefty, elbow=epositive, wrist=wpositive, fatherId=fReference[0]}
  [893] = {x=11.108, y=0.000, z=-7.046, rx=-0.000, ry=0.000, rz=-0.000, shoulder=lefty, elbow=epositive, wrist=wpositive, fatherId=fReference[0]}
  [894] = {x=11.616, y=0.000, z=-7.055, rx=-0.000, ry=0.000, rz=-0.000, shoulder=lefty, elbow=epositive, wrist=wpositive, fatherId=fReference[0]}
  [895] = {x=12.125, y=0.000, z=-7.064, rx=-0.000, ry=0.000, rz=-0.000, shoulder=lefty, elbow=epositive, wrist=wpositive, fatherId=fReference[0]}
  [896] = {x=12.632, y=0.000, z=-7.074, rx=-0.000, ry=0.000, rz=-0.000, shoulder=lefty, elbow=epositive, wrist=wpositive, fatherId=fReference[0]}
  [897] = {x=13.140, y=0.000, z=-7.084, rx=-0.000, ry=0.000, rz=-0.000, shoulder=lefty, elbow=epositive, wrist=wpositive, fatherId=fReference[0]}
  [898] = {x=13.650, y=0.000, z=-7.093, rx=-0.000, ry=0.000, rz=-0.000, shoulder=lefty, elbow=epositive, wrist=wpositive, fatherId=fReference[0]}
  [899] = {x=14.158, y=0.000, z=-7.103, rx=-0.000, ry=0.000, rz=-0.000, shoulder=lefty, elbow=epositive, wrist=wpositive, fatherId=fReference[0]}
  [900] = {x=14.667, y=0.000, z=-7.112, rx=-0.000, ry=0.000, rz=-0.000, shoulder=lefty, elbow=epositive, wrist=wpositive, fatherId=fReference[0]}
  [901] = {x=15.175, y=0.000, z=-7.122, rx=-0.000, ry=0.000, rz=-0.000, shoulder=lefty, elbow=epositive, wrist=wpositive, fatherId=fReference[0]}
  [902] = {x=15.685, y=0.000, z=-7.130, rx=-0.000, ry=0.000, rz=-0.000, shoulder=lefty, elbow=epositive, wrist=wpositive, fatherId=fReference[0]}
  [903] = {x=16.194, y=0.000, z=-7.141, rx=-0.000, ry=0.000, rz=-0.000, shoulder=lefty, elbow=epositive, wrist=wpositive, fatherId=fReference[0]}
  [904] = {x=16.704, y=0.000, z=-7.150, rx=-0.000, ry=0.000, rz=-0.000, shoulder=lefty, elbow=epositive, wrist=wpositive, fatherId=fReference[0]}
  [905] = {x=17.213, y=0.000, z=-7.160, rx=-0.000, ry=0.000, rz=-0.000, shoulder=lefty, elbow=epositive, wrist=wpositive, fatherId=fReference[0]}
  [906] = {x=17.723, y=0.000, z=-7.169, rx=-0.000, ry=0.000, rz=-0.000, shoulder=lefty, elbow=epositive, wrist=wpositive, fatherId=fReference[0]}
  [907] = {x=18.234, y=0.000, z=-7.179, rx=-0.000, ry=0.000, rz=-0.000, shoulder=lefty, elbow=epositive, wrist=wpositive, fatherId=fReference[0]}
  [908] = {x=18.744, y=0.000, z=-7.190, rx=-0.000, ry=0.000, rz=-0.000, shoulder=lefty, elbow=epositive, wrist=wpositive, fatherId=fReference[0]}
  [909] = {x=19.254, y=0.000, z=-7.199, rx=-0.000, ry=0.000, rz=-0.000, shoulder=lefty, elbow=epositive, wrist=wpositive, fatherId=fReference[0]}
  [910] = {x=19.764, y=0.000, z=-7.209, rx=-0.000, ry=0.000, rz=-0.000, shoulder=lefty, elbow=epositive, wrist=wpositive, fatherId=fReference[0]}
  [911] = {x=20.277, y=0.000, z=-7.219, rx=-0.000, ry=0.000, rz=-0.000, shoulder=lefty, elbow=epositive, wrist=wpositive, fatherId=fReference[0]}
  [912] = {x=20.787, y=0.000, z=-7.228, rx=-0.000, ry=0.000, rz=-0.000, shoulder=lefty, elbow=epositive, wrist=wpositive, fatherId=fReference[0]}
  [913] = {x=21.299, y=0.000, z=-7.239, rx=-0.000, ry=0.000, rz=-0.000, shoulder=lefty, elbow=epositive, wrist=wpositive, fatherId=fReference[0]}
  [914] = {x=21.811, y=0.000, z=-7.247, rx=-0.000, ry=0.000, rz=-0.000, shoulder=lefty, elbow=epositive, wrist=wpositive, fatherId=fReference[0]}
  [915] = {x=22.323, y=0.000, z=-7.258, rx=-0.000, ry=0.000, rz=-0.000, shoulder=lefty, elbow=epositive, wrist=wpositive, fatherId=fReference[0]}
  [916] = {x=22.835, y=0.000, z=-7.269, rx=-0.000, ry=0.000, rz=-0.000, shoulder=lefty, elbow=epositive, wrist=wpositive, fatherId=fReference[0]}
  [917] = {x=23.348, y=0.000, z=-7.279, rx=-0.000, ry=0.000, rz=-0.000, shoulder=lefty, elbow=epositive, wrist=wpositive, fatherId=fReference[0]}
  [918] = {x=23.861, y=0.000, z=-7.289, rx=-0.000, ry=0.000, rz=-0.000, shoulder=lefty, elbow=epositive, wrist=wpositive, fatherId=fReference[0]}
  [919] = {x=24.372, y=0.000, z=-7.296, rx=-0.000, ry=0.000, rz=-0.000, shoulder=lefty, elbow=epositive, wrist=wpositive, fatherId=fReference[0]}
  [920] = {x=24.887, y=0.000, z=-7.308, rx=-0.000, ry=0.000, rz=-0.000, shoulder=lefty, elbow=epositive, wrist=wpositive, fatherId=fReference[0]}
  [921] = {x=25.399, y=0.000, z=-7.316, rx=-0.000, ry=0.000, rz=-0.000, shoulder=lefty, elbow=epositive, wrist=wpositive, fatherId=fReference[0]}
  [922] = {x=25.915, y=0.000, z=-7.327, rx=-0.000, ry=0.000, rz=-0.000, shoulder=lefty, elbow=epositive, wrist=wpositive, fatherId=fReference[0]}
  [923] = {x=26.429, y=0.000, z=-7.338, rx=-0.000, ry=0.000, rz=-0.000, shoulder=lefty, elbow=epositive, wrist=wpositive, fatherId=fReference[0]}
  [924] = {x=26.945, y=0.000, z=-7.348, rx=-0.000, ry=0.000, rz=-0.000, shoulder=lefty, elbow=epositive, wrist=wpositive, fatherId=fReference[0]}
  [925] = {x=27.460, y=0.000, z=-7.358, rx=-0.000, ry=0.000, rz=-0.000, shoulder=lefty, elbow=epositive, wrist=wpositive, fatherId=fReference[0]}
  [926] = {x=27.976, y=0.000, z=-7.366, rx=-0.000, ry=0.000, rz=-0.000, shoulder=lefty, elbow=epositive, wrist=wpositive, fatherId=fReference[0]}
  [927] = {x=28.493, y=0.000, z=-7.375, rx=-0.000, ry=0.000, rz=-0.000, shoulder=lefty, elbow=epositive, wrist=wpositive, fatherId=fReference[0]}
  [928] = {x=29.013, y=0.000, z=-7.386, rx=-0.000, ry=0.000, rz=-0.000, shoulder=lefty, elbow=epositive, wrist=wpositive, fatherId=fReference[0]}
  [929] = {x=29.534, y=0.000, z=-7.396, rx=-0.000, ry=0.000, rz=-0.000, shoulder=lefty, elbow=epositive, wrist=wpositive, fatherId=fReference[0]}
  [930] = {x=30.056, y=0.000, z=-7.408, rx=-0.000, ry=0.000, rz=-0.000, shoulder=lefty, elbow=epositive, wrist=wpositive, fatherId=fReference[0]}
  [931] = {x=30.582, y=0.000, z=-7.419, rx=-0.000, ry=0.000, rz=-0.000, shoulder=lefty, elbow=epositive, wrist=wpositive, fatherId=fReference[0]}
  [932] = {x=31.109, y=0.000, z=-7.430, rx=-0.000, ry=0.000, rz=-0.000, shoulder=lefty, elbow=epositive, wrist=wpositive, fatherId=fReference[0]}
  [933] = {x=31.643, y=0.000, z=-7.440, rx=-0.000, ry=0.000, rz=-0.000, shoulder=lefty, elbow=epositive, wrist=wpositive, fatherId=fReference[0]}
  [934] = {x=32.176, y=0.000, z=-7.451, rx=-0.000, ry=0.000, rz=-0.000, shoulder=lefty, elbow=epositive, wrist=wpositive, fatherId=fReference[0]}
  [935] = {x=32.713, y=0.000, z=-7.461, rx=-0.000, ry=0.000, rz=-0.000, shoulder=lefty, elbow=epositive, wrist=wpositive, fatherId=fReference[0]}
  [936] = {x=33.254, y=0.000, z=-7.472, rx=-0.000, ry=0.000, rz=-0.000, shoulder=lefty, elbow=epositive, wrist=wpositive, fatherId=fReference[0]}
  [937] = {x=33.795, y=0.000, z=-7.477, rx=-0.000, ry=0.000, rz=-0.000, shoulder=lefty, elbow=epositive, wrist=wpositive, fatherId=fReference[0]}
  [938] = {x=34.339, y=0.000, z=-7.483, rx=-0.000, ry=0.000, rz=-0.000, shoulder=lefty, elbow=epositive, wrist=wpositive, fatherId=fReference[0]}
  [939] = {x=33.040, y=0.000, z=-7.506, rx=-0.000, ry=0.000, rz=-0.000, shoulder=lefty, elbow=epositive, wrist=wpositive, fatherId=fReference[0]}
  [940] = {x=32.384, y=0.000, z=-7.498, rx=-0.000, ry=0.000, rz=-0.000, shoulder=lefty, elbow=epositive, wrist=wpositive, fatherId=fReference[0]}
  [941] = {x=31.801, y=0.000, z=-7.494, rx=-0.000, ry=0.000, rz=-0.000, shoulder=lefty, elbow=epositive, wrist=wpositive, fatherId=fReference[0]}
  [942] = {x=31.256, y=0.000, z=-7.494, rx=-0.000, ry=0.000, rz=-0.000, shoulder=lefty, elbow=epositive, wrist=wpositive, fatherId=fReference[0]}
  [943] = {x=30.729, y=0.000, z=-7.496, rx=-0.000, ry=0.000, rz=-0.000, shoulder=lefty, elbow=epositive, wrist=wpositive, fatherId=fReference[0]}
  [944] = {x=30.207, y=0.000, z=-7.499, rx=-0.000, ry=0.000, rz=-0.000, shoulder=lefty, elbow=epositive, wrist=wpositive, fatherId=fReference[0]}
  [945] = {x=29.690, y=0.000, z=-7.504, rx=-0.000, ry=0.000, rz=-0.000, shoulder=lefty, elbow=epositive, wrist=wpositive, fatherId=fReference[0]}
  [946] = {x=29.176, y=0.000, z=-7.510, rx=-0.000, ry=0.000, rz=-0.000, shoulder=lefty, elbow=epositive, wrist=wpositive, fatherId=fReference[0]}
  [947] = {x=28.665, y=0.000, z=-7.516, rx=-0.000, ry=0.000, rz=-0.000, shoulder=lefty, elbow=epositive, wrist=wpositive, fatherId=fReference[0]}
  [948] = {x=28.154, y=0.000, z=-7.523, rx=-0.000, ry=0.000, rz=-0.000, shoulder=lefty, elbow=epositive, wrist=wpositive, fatherId=fReference[0]}
  [949] = {x=27.647, y=0.000, z=-7.530, rx=-0.000, ry=0.000, rz=-0.000, shoulder=lefty, elbow=epositive, wrist=wpositive, fatherId=fReference[0]}
  [950] = {x=27.144, y=0.000, z=-7.538, rx=-0.000, ry=0.000, rz=-0.000, shoulder=lefty, elbow=epositive, wrist=wpositive, fatherId=fReference[0]}
  [951] = {x=26.641, y=0.000, z=-7.545, rx=-0.000, ry=0.000, rz=-0.000, shoulder=lefty, elbow=epositive, wrist=wpositive, fatherId=fReference[0]}
  [952] = {x=26.137, y=0.000, z=-7.553, rx=-0.000, ry=0.000, rz=-0.000, shoulder=lefty, elbow=epositive, wrist=wpositive, fatherId=fReference[0]}
  [953] = {x=25.633, y=0.000, z=-7.560, rx=-0.000, ry=0.000, rz=-0.000, shoulder=lefty, elbow=epositive, wrist=wpositive, fatherId=fReference[0]}
  [954] = {x=25.130, y=0.000, z=-7.569, rx=-0.000, ry=0.000, rz=-0.000, shoulder=lefty, elbow=epositive, wrist=wpositive, fatherId=fReference[0]}
  [955] = {x=24.627, y=0.000, z=-7.577, rx=-0.000, ry=0.000, rz=-0.000, shoulder=lefty, elbow=epositive, wrist=wpositive, fatherId=fReference[0]}
  [956] = {x=24.126, y=0.000, z=-7.587, rx=-0.000, ry=0.000, rz=-0.000, shoulder=lefty, elbow=epositive, wrist=wpositive, fatherId=fReference[0]}
  [957] = {x=23.628, y=0.000, z=-7.596, rx=-0.000, ry=0.000, rz=-0.000, shoulder=lefty, elbow=epositive, wrist=wpositive, fatherId=fReference[0]}
  [958] = {x=23.131, y=0.000, z=-7.605, rx=-0.000, ry=0.000, rz=-0.000, shoulder=lefty, elbow=epositive, wrist=wpositive, fatherId=fReference[0]}
  [959] = {x=22.632, y=0.000, z=-7.613, rx=-0.000, ry=0.000, rz=-0.000, shoulder=lefty, elbow=epositive, wrist=wpositive, fatherId=fReference[0]}
  [960] = {x=22.132, y=0.000, z=-7.622, rx=-0.000, ry=0.000, rz=-0.000, shoulder=lefty, elbow=epositive, wrist=wpositive, fatherId=fReference[0]}
  [961] = {x=21.632, y=0.000, z=-7.631, rx=-0.000, ry=0.000, rz=-0.000, shoulder=lefty, elbow=epositive, wrist=wpositive, fatherId=fReference[0]}
  [962] = {x=21.133, y=0.000, z=-7.640, rx=-0.000, ry=0.000, rz=-0.000, shoulder=lefty, elbow=epositive, wrist=wpositive, fatherId=fReference[0]}
  [963] = {x=20.633, y=0.000, z=-7.649, rx=-0.000, ry=0.000, rz=-0.000, shoulder=lefty, elbow=epositive, wrist=wpositive, fatherId=fReference[0]}
  [964] = {x=20.135, y=0.000, z=-7.658, rx=-0.000, ry=0.000, rz=-0.000, shoulder=lefty, elbow=epositive, wrist=wpositive, fatherId=fReference[0]}
  [965] = {x=19.637, y=0.000, z=-7.668, rx=-0.000, ry=0.000, rz=-0.000, shoulder=lefty, elbow=epositive, wrist=wpositive, fatherId=fReference[0]}
  [966] = {x=19.139, y=0.000, z=-7.677, rx=-0.000, ry=0.000, rz=-0.000, shoulder=lefty, elbow=epositive, wrist=wpositive, fatherId=fReference[0]}
  [967] = {x=18.643, y=0.000, z=-7.687, rx=-0.000, ry=0.000, rz=-0.000, shoulder=lefty, elbow=epositive, wrist=wpositive, fatherId=fReference[0]}
  [968] = {x=18.143, y=0.000, z=-7.696, rx=-0.000, ry=0.000, rz=-0.000, shoulder=lefty, elbow=epositive, wrist=wpositive, fatherId=fReference[0]}
  [969] = {x=17.644, y=0.000, z=-7.705, rx=-0.000, ry=0.000, rz=-0.000, shoulder=lefty, elbow=epositive, wrist=wpositive, fatherId=fReference[0]}
  [970] = {x=17.149, y=0.000, z=-7.715, rx=-0.000, ry=0.000, rz=-0.000, shoulder=lefty, elbow=epositive, wrist=wpositive, fatherId=fReference[0]}
  [971] = {x=16.650, y=0.000, z=-7.724, rx=-0.000, ry=0.000, rz=-0.000, shoulder=lefty, elbow=epositive, wrist=wpositive, fatherId=fReference[0]}
  [972] = {x=16.151, y=0.000, z=-7.734, rx=-0.000, ry=0.000, rz=-0.000, shoulder=lefty, elbow=epositive, wrist=wpositive, fatherId=fReference[0]}
  [973] = {x=15.652, y=0.000, z=-7.743, rx=-0.000, ry=0.000, rz=-0.000, shoulder=lefty, elbow=epositive, wrist=wpositive, fatherId=fReference[0]}
  [974] = {x=15.154, y=0.000, z=-7.753, rx=-0.000, ry=0.000, rz=-0.000, shoulder=lefty, elbow=epositive, wrist=wpositive, fatherId=fReference[0]}
  [975] = {x=14.656, y=0.000, z=-7.762, rx=-0.000, ry=0.000, rz=-0.000, shoulder=lefty, elbow=epositive, wrist=wpositive, fatherId=fReference[0]}
  [976] = {x=14.160, y=0.000, z=-7.772, rx=-0.000, ry=0.000, rz=-0.000, shoulder=lefty, elbow=epositive, wrist=wpositive, fatherId=fReference[0]}
  [977] = {x=13.661, y=0.000, z=-7.781, rx=-0.000, ry=0.000, rz=-0.000, shoulder=lefty, elbow=epositive, wrist=wpositive, fatherId=fReference[0]}
  [978] = {x=13.163, y=0.000, z=-7.791, rx=-0.000, ry=0.000, rz=-0.000, shoulder=lefty, elbow=epositive, wrist=wpositive, fatherId=fReference[0]}
  [979] = {x=12.665, y=0.000, z=-7.800, rx=-0.000, ry=0.000, rz=-0.000, shoulder=lefty, elbow=epositive, wrist=wpositive, fatherId=fReference[0]}
  [980] = {x=12.166, y=0.000, z=-7.809, rx=-0.000, ry=0.000, rz=-0.000, shoulder=lefty, elbow=epositive, wrist=wpositive, fatherId=fReference[0]}
  [981] = {x=11.666, y=0.000, z=-7.819, rx=-0.000, ry=0.000, rz=-0.000, shoulder=lefty, elbow=epositive, wrist=wpositive, fatherId=fReference[0]}
  [982] = {x=11.166, y=0.000, z=-7.828, rx=-0.000, ry=0.000, rz=-0.000, shoulder=lefty, elbow=epositive, wrist=wpositive, fatherId=fReference[0]}
  [983] = {x=10.665, y=0.000, z=-7.837, rx=-0.000, ry=0.000, rz=-0.000, shoulder=lefty, elbow=epositive, wrist=wpositive, fatherId=fReference[0]}
  [984] = {x=10.163, y=0.000, z=-7.846, rx=-0.000, ry=0.000, rz=-0.000, shoulder=lefty, elbow=epositive, wrist=wpositive, fatherId=fReference[0]}
  [985] = {x=9.662, y=0.000, z=-7.855, rx=-0.000, ry=0.000, rz=-0.000, shoulder=lefty, elbow=epositive, wrist=wpositive, fatherId=fReference[0]}
  [986] = {x=9.161, y=0.000, z=-7.864, rx=-0.000, ry=0.000, rz=-0.000, shoulder=lefty, elbow=epositive, wrist=wpositive, fatherId=fReference[0]}
  [987] = {x=8.660, y=0.000, z=-7.873, rx=-0.000, ry=0.000, rz=-0.000, shoulder=lefty, elbow=epositive, wrist=wpositive, fatherId=fReference[0]}
  [988] = {x=8.157, y=0.000, z=-7.882, rx=-0.000, ry=0.000, rz=-0.000, shoulder=lefty, elbow=epositive, wrist=wpositive, fatherId=fReference[0]}
  [989] = {x=7.650, y=0.000, z=-7.891, rx=-0.000, ry=0.000, rz=-0.000, shoulder=lefty, elbow=epositive, wrist=wpositive, fatherId=fReference[0]}
  [990] = {x=7.145, y=0.000, z=-7.899, rx=-0.000, ry=0.000, rz=-0.000, shoulder=lefty, elbow=epositive, wrist=wpositive, fatherId=fReference[0]}
  [991] = {x=6.635, y=0.000, z=-7.906, rx=-0.000, ry=0.000, rz=-0.000, shoulder=lefty, elbow=epositive, wrist=wpositive, fatherId=fReference[0]}
  [992] = {x=6.128, y=0.000, z=-7.914, rx=-0.000, ry=0.000, rz=-0.000, shoulder=lefty, elbow=epositive, wrist=wpositive, fatherId=fReference[0]}
  [993] = {x=5.621, y=0.000, z=-7.922, rx=-0.000, ry=0.000, rz=-0.000, shoulder=lefty, elbow=epositive, wrist=wpositive, fatherId=fReference[0]}
  [994] = {x=5.117, y=0.000, z=-7.930, rx=-0.000, ry=0.000, rz=-0.000, shoulder=lefty, elbow=epositive, wrist=wpositive, fatherId=fReference[0]}
  [995] = {x=4.610, y=0.000, z=-7.939, rx=-0.000, ry=0.000, rz=-0.000, shoulder=lefty, elbow=epositive, wrist=wpositive, fatherId=fReference[0]}
  [996] = {x=4.104, y=0.000, z=-7.947, rx=-0.000, ry=0.000, rz=-0.000, shoulder=lefty, elbow=epositive, wrist=wpositive, fatherId=fReference[0]}
  [997] = {x=3.599, y=0.000, z=-7.955, rx=-0.000, ry=0.000, rz=-0.000, shoulder=lefty, elbow=epositive, wrist=wpositive, fatherId=fReference[0]}
  [998] = {x=3.092, y=0.000, z=-7.964, rx=-0.000, ry=0.000, rz=-0.000, shoulder=lefty, elbow=epositive, wrist=wpositive, fatherId=fReference[0]}
  [999] = {x=2.586, y=0.000, z=-7.973, rx=-0.000, ry=0.000, rz=-0.000, shoulder=lefty, elbow=epositive, wrist=wpositive, fatherId=fReference[0]}
  [1000] = {x=2.082, y=0.000, z=-7.982, rx=-0.000, ry=0.000, rz=-0.000, shoulder=lefty, elbow=epositive, wrist=wpositive, fatherId=fReference[0]}
  [1001] = {x=1.579, y=0.000, z=-7.991, rx=-0.000, ry=0.000, rz=-0.000, shoulder=lefty, elbow=epositive, wrist=wpositive, fatherId=fReference[0]}
  [1002] = {x=1.075, y=0.000, z=-8.000, rx=-0.000, ry=0.000, rz=-0.000, shoulder=lefty, elbow=epositive, wrist=wpositive, fatherId=fReference[0]}
  [1003] = {x=0.570, y=0.000, z=-8.009, rx=-0.000, ry=0.000, rz=-0.000, shoulder=lefty, elbow=epositive, wrist=wpositive, fatherId=fReference[0]}
  [1004] = {x=0.067, y=0.000, z=-8.019, rx=-0.000, ry=0.000, rz=-0.000, shoulder=lefty, elbow=epositive, wrist=wpositive, fatherId=fReference[0]}
  [1005] = {x=-0.435, y=0.000, z=-8.028, rx=-0.000, ry=0.000, rz=-0.000, shoulder=lefty, elbow=epositive, wrist=wpositive, fatherId=fReference[0]}
  [1006] = {x=-0.936, y=0.000, z=-8.038, rx=-0.000, ry=0.000, rz=-0.000, shoulder=lefty, elbow=epositive, wrist=wpositive, fatherId=fReference[0]}
  [1007] = {x=-1.437, y=0.000, z=-8.048, rx=-0.000, ry=0.000, rz=-0.000, shoulder=lefty, elbow=epositive, wrist=wpositive, fatherId=fReference[0]}
  [1008] = {x=-1.939, y=0.000, z=-8.057, rx=-0.000, ry=0.000, rz=-0.000, shoulder=lefty, elbow=epositive, wrist=wpositive, fatherId=fReference[0]}
  [1009] = {x=-2.439, y=0.000, z=-8.067, rx=-0.000, ry=0.000, rz=-0.000, shoulder=lefty, elbow=epositive, wrist=wpositive, fatherId=fReference[0]}
  [1010] = {x=-2.939, y=0.000, z=-8.076, rx=-0.000, ry=0.000, rz=-0.000, shoulder=lefty, elbow=epositive, wrist=wpositive, fatherId=fReference[0]}
  [1011] = {x=-3.439, y=0.000, z=-8.086, rx=-0.000, ry=0.000, rz=-0.000, shoulder=lefty, elbow=epositive, wrist=wpositive, fatherId=fReference[0]}
  [1012] = {x=-3.935, y=0.000, z=-8.096, rx=-0.000, ry=0.000, rz=-0.000, shoulder=lefty, elbow=epositive, wrist=wpositive, fatherId=fReference[0]}
  [1013] = {x=-4.437, y=0.000, z=-8.106, rx=-0.000, ry=0.000, rz=-0.000, shoulder=lefty, elbow=epositive, wrist=wpositive, fatherId=fReference[0]}
  [1014] = {x=-4.933, y=0.000, z=-8.115, rx=-0.000, ry=0.000, rz=-0.000, shoulder=lefty, elbow=epositive, wrist=wpositive, fatherId=fReference[0]}
  [1015] = {x=-5.434, y=0.000, z=-8.125, rx=-0.000, ry=0.000, rz=-0.000, shoulder=lefty, elbow=epositive, wrist=wpositive, fatherId=fReference[0]}
  [1016] = {x=-5.935, y=0.000, z=-8.135, rx=-0.000, ry=0.000, rz=-0.000, shoulder=lefty, elbow=epositive, wrist=wpositive, fatherId=fReference[0]}
  [1017] = {x=-6.429, y=0.000, z=-8.145, rx=-0.000, ry=0.000, rz=-0.000, shoulder=lefty, elbow=epositive, wrist=wpositive, fatherId=fReference[0]}
  [1018] = {x=-6.931, y=0.000, z=-8.155, rx=-0.000, ry=0.000, rz=-0.000, shoulder=lefty, elbow=epositive, wrist=wpositive, fatherId=fReference[0]}
  [1019] = {x=-7.426, y=0.000, z=-8.165, rx=-0.000, ry=0.000, rz=-0.000, shoulder=lefty, elbow=epositive, wrist=wpositive, fatherId=fReference[0]}
  [1020] = {x=-7.929, y=0.000, z=-8.174, rx=-0.000, ry=0.000, rz=-0.000, shoulder=lefty, elbow=epositive, wrist=wpositive, fatherId=fReference[0]}
  [1021] = {x=-8.424, y=0.000, z=-8.184, rx=-0.000, ry=0.000, rz=-0.000, shoulder=lefty, elbow=epositive, wrist=wpositive, fatherId=fReference[0]}
  [1022] = {x=-8.926, y=0.000, z=-8.194, rx=-0.000, ry=0.000, rz=-0.000, shoulder=lefty, elbow=epositive, wrist=wpositive, fatherId=fReference[0]}
  [1023] = {x=-9.421, y=0.000, z=-8.204, rx=-0.000, ry=0.000, rz=-0.000, shoulder=lefty, elbow=epositive, wrist=wpositive, fatherId=fReference[0]}
  [1024] = {x=-9.924, y=0.000, z=-8.214, rx=-0.000, ry=0.000, rz=-0.000, shoulder=lefty, elbow=epositive, wrist=wpositive, fatherId=fReference[0]}
  [1025] = {x=-10.420, y=0.000, z=-8.224, rx=-0.000, ry=0.000, rz=-0.000, shoulder=lefty, elbow=epositive, wrist=wpositive, fatherId=fReference[0]}
  [1026] = {x=-10.922, y=0.000, z=-8.234, rx=-0.000, ry=0.000, rz=-0.000, shoulder=lefty, elbow=epositive, wrist=wpositive, fatherId=fReference[0]}
  [1027] = {x=-11.424, y=0.000, z=-8.243, rx=-0.000, ry=0.000, rz=-0.000, shoulder=lefty, elbow=epositive, wrist=wpositive, fatherId=fReference[0]}
  [1028] = {x=-11.920, y=0.000, z=-8.254, rx=-0.000, ry=0.000, rz=-0.000, shoulder=lefty, elbow=epositive, wrist=wpositive, fatherId=fReference[0]}
  [1029] = {x=-12.424, y=0.000, z=-8.263, rx=-0.000, ry=0.000, rz=-0.000, shoulder=lefty, elbow=epositive, wrist=wpositive, fatherId=fReference[0]}
  [1030] = {x=-12.920, y=0.000, z=-8.274, rx=-0.000, ry=0.000, rz=-0.000, shoulder=lefty, elbow=epositive, wrist=wpositive, fatherId=fReference[0]}
  [1031] = {x=-13.425, y=0.000, z=-8.283, rx=-0.000, ry=0.000, rz=-0.000, shoulder=lefty, elbow=epositive, wrist=wpositive, fatherId=fReference[0]}
  [1032] = {x=-13.924, y=0.000, z=-8.293, rx=-0.000, ry=0.000, rz=-0.000, shoulder=lefty, elbow=epositive, wrist=wpositive, fatherId=fReference[0]}
  [1033] = {x=-14.428, y=0.000, z=-8.303, rx=-0.000, ry=0.000, rz=-0.000, shoulder=lefty, elbow=epositive, wrist=wpositive, fatherId=fReference[0]}
  [1034] = {x=-14.932, y=0.000, z=-8.313, rx=-0.000, ry=0.000, rz=-0.000, shoulder=lefty, elbow=epositive, wrist=wpositive, fatherId=fReference[0]}
  [1035] = {x=-15.434, y=0.000, z=-8.322, rx=-0.000, ry=0.000, rz=-0.000, shoulder=lefty, elbow=epositive, wrist=wpositive, fatherId=fReference[0]}
  [1036] = {x=-15.935, y=0.000, z=-8.333, rx=-0.000, ry=0.000, rz=-0.000, shoulder=lefty, elbow=epositive, wrist=wpositive, fatherId=fReference[0]}
  [1037] = {x=-16.437, y=0.000, z=-8.343, rx=-0.000, ry=0.000, rz=-0.000, shoulder=lefty, elbow=epositive, wrist=wpositive, fatherId=fReference[0]}
  [1038] = {x=-16.938, y=0.000, z=-8.354, rx=-0.000, ry=0.000, rz=-0.000, shoulder=lefty, elbow=epositive, wrist=wpositive, fatherId=fReference[0]}
  [1039] = {x=-17.438, y=0.000, z=-8.364, rx=-0.000, ry=0.000, rz=-0.000, shoulder=lefty, elbow=epositive, wrist=wpositive, fatherId=fReference[0]}
  [1040] = {x=-17.935, y=0.000, z=-8.375, rx=-0.000, ry=0.000, rz=-0.000, shoulder=lefty, elbow=epositive, wrist=wpositive, fatherId=fReference[0]}
  [1041] = {x=-18.435, y=0.000, z=-8.387, rx=-0.000, ry=0.000, rz=-0.000, shoulder=lefty, elbow=epositive, wrist=wpositive, fatherId=fReference[0]}
  [1042] = {x=-18.935, y=0.000, z=-8.398, rx=-0.000, ry=0.000, rz=-0.000, shoulder=lefty, elbow=epositive, wrist=wpositive, fatherId=fReference[0]}
  [1043] = {x=-19.434, y=0.000, z=-8.409, rx=-0.000, ry=0.000, rz=-0.000, shoulder=lefty, elbow=epositive, wrist=wpositive, fatherId=fReference[0]}
  [1044] = {x=-19.936, y=0.000, z=-8.420, rx=-0.000, ry=0.000, rz=-0.000, shoulder=lefty, elbow=epositive, wrist=wpositive, fatherId=fReference[0]}
  [1045] = {x=-20.433, y=0.000, z=-8.431, rx=-0.000, ry=0.000, rz=-0.000, shoulder=lefty, elbow=epositive, wrist=wpositive, fatherId=fReference[0]}
  [1046] = {x=-20.935, y=0.000, z=-8.443, rx=-0.000, ry=0.000, rz=-0.000, shoulder=lefty, elbow=epositive, wrist=wpositive, fatherId=fReference[0]}
  [1047] = {x=-21.433, y=0.000, z=-8.454, rx=-0.000, ry=0.000, rz=-0.000, shoulder=lefty, elbow=epositive, wrist=wpositive, fatherId=fReference[0]}
  [1048] = {x=-21.930, y=0.000, z=-8.466, rx=-0.000, ry=0.000, rz=-0.000, shoulder=lefty, elbow=epositive, wrist=wpositive, fatherId=fReference[0]}
  [1049] = {x=-22.431, y=0.000, z=-8.479, rx=-0.000, ry=0.000, rz=-0.000, shoulder=lefty, elbow=epositive, wrist=wpositive, fatherId=fReference[0]}
  [1050] = {x=-22.930, y=0.000, z=-8.491, rx=-0.000, ry=0.000, rz=-0.000, shoulder=lefty, elbow=epositive, wrist=wpositive, fatherId=fReference[0]}
  [1051] = {x=-23.432, y=0.000, z=-8.503, rx=-0.000, ry=0.000, rz=-0.000, shoulder=lefty, elbow=epositive, wrist=wpositive, fatherId=fReference[0]}
  [1052] = {x=-23.932, y=0.000, z=-8.515, rx=-0.000, ry=0.000, rz=-0.000, shoulder=lefty, elbow=epositive, wrist=wpositive, fatherId=fReference[0]}
  [1053] = {x=-24.432, y=0.000, z=-8.527, rx=-0.000, ry=0.000, rz=-0.000, shoulder=lefty, elbow=epositive, wrist=wpositive, fatherId=fReference[0]}
  [1054] = {x=-24.933, y=0.000, z=-8.540, rx=-0.000, ry=0.000, rz=-0.000, shoulder=lefty, elbow=epositive, wrist=wpositive, fatherId=fReference[0]}
  [1055] = {x=-25.432, y=0.000, z=-8.553, rx=-0.000, ry=0.000, rz=-0.000, shoulder=lefty, elbow=epositive, wrist=wpositive, fatherId=fReference[0]}
  [1056] = {x=-25.930, y=0.000, z=-8.568, rx=-0.000, ry=0.000, rz=-0.000, shoulder=lefty, elbow=epositive, wrist=wpositive, fatherId=fReference[0]}
  [1057] = {x=-26.421, y=0.000, z=-8.584, rx=-0.000, ry=0.000, rz=-0.000, shoulder=lefty, elbow=epositive, wrist=wpositive, fatherId=fReference[0]}
  [1058] = {x=-26.914, y=0.000, z=-8.601, rx=-0.000, ry=0.000, rz=-0.000, shoulder=lefty, elbow=epositive, wrist=wpositive, fatherId=fReference[0]}
  [1059] = {x=-27.408, y=0.000, z=-8.618, rx=-0.000, ry=0.000, rz=-0.000, shoulder=lefty, elbow=epositive, wrist=wpositive, fatherId=fReference[0]}
  [1060] = {x=-27.906, y=0.000, z=-8.636, rx=-0.000, ry=0.000, rz=-0.000, shoulder=lefty, elbow=epositive, wrist=wpositive, fatherId=fReference[0]}
  [1061] = {x=-28.406, y=0.000, z=-8.655, rx=-0.000, ry=0.000, rz=-0.000, shoulder=lefty, elbow=epositive, wrist=wpositive, fatherId=fReference[0]}
  [1062] = {x=-28.927, y=0.000, z=-8.675, rx=-0.000, ry=0.000, rz=-0.000, shoulder=lefty, elbow=epositive, wrist=wpositive, fatherId=fReference[0]}
  [1063] = {x=-29.460, y=0.000, z=-8.694, rx=-0.000, ry=0.000, rz=-0.000, shoulder=lefty, elbow=epositive, wrist=wpositive, fatherId=fReference[0]}
  [1064] = {x=-30.007, y=0.000, z=-8.709, rx=-0.000, ry=0.000, rz=-0.000, shoulder=lefty, elbow=epositive, wrist=wpositive, fatherId=fReference[0]}
  [1065] = {x=-28.841, y=0.000, z=-8.593, rx=-0.000, ry=0.000, rz=-0.000, shoulder=lefty, elbow=epositive, wrist=wpositive, fatherId=fReference[0]}
  [1066] = {x=-28.333, y=0.000, z=-8.558, rx=-0.000, ry=0.000, rz=-0.000, shoulder=lefty, elbow=epositive, wrist=wpositive, fatherId=fReference[0]}
  [1067] = {x=-27.860, y=0.000, z=-8.544, rx=-0.000, ry=0.000, rz=-0.000, shoulder=lefty, elbow=epositive, wrist=wpositive, fatherId=fReference[0]}
  [1068] = {x=-27.388, y=0.000, z=-8.534, rx=-0.000, ry=0.000, rz=-0.000, shoulder=lefty, elbow=epositive, wrist=wpositive, fatherId=fReference[0]}
  [1069] = {x=-26.912, y=0.000, z=-8.528, rx=-0.000, ry=0.000, rz=-0.000, shoulder=lefty, elbow=epositive, wrist=wpositive, fatherId=fReference[0]}
  [1070] = {x=-26.431, y=0.000, z=-8.526, rx=-0.000, ry=0.000, rz=-0.000, shoulder=lefty, elbow=epositive, wrist=wpositive, fatherId=fReference[0]}
  [1071] = {x=-25.938, y=0.000, z=-8.527, rx=-0.000, ry=0.000, rz=-0.000, shoulder=lefty, elbow=epositive, wrist=wpositive, fatherId=fReference[0]}
  [1072] = {x=-25.442, y=0.000, z=-8.530, rx=-0.000, ry=0.000, rz=-0.000, shoulder=lefty, elbow=epositive, wrist=wpositive, fatherId=fReference[0]}
  [1073] = {x=-24.943, y=0.000, z=-8.534, rx=-0.000, ry=0.000, rz=-0.000, shoulder=lefty, elbow=epositive, wrist=wpositive, fatherId=fReference[0]}
  [1074] = {x=-24.443, y=0.000, z=-8.539, rx=-0.000, ry=0.000, rz=-0.000, shoulder=lefty, elbow=epositive, wrist=wpositive, fatherId=fReference[0]}
  [1075] = {x=-23.942, y=0.000, z=-8.546, rx=-0.000, ry=0.000, rz=-0.000, shoulder=lefty, elbow=epositive, wrist=wpositive, fatherId=fReference[0]}
  [1076] = {x=-23.439, y=0.000, z=-8.553, rx=-0.000, ry=0.000, rz=-0.000, shoulder=lefty, elbow=epositive, wrist=wpositive, fatherId=fReference[0]}
  [1077] = {x=-22.937, y=0.000, z=-8.560, rx=-0.000, ry=0.000, rz=-0.000, shoulder=lefty, elbow=epositive, wrist=wpositive, fatherId=fReference[0]}
  [1078] = {x=-22.433, y=0.000, z=-8.568, rx=-0.000, ry=0.000, rz=-0.000, shoulder=lefty, elbow=epositive, wrist=wpositive, fatherId=fReference[0]}
  [1079] = {x=-21.926, y=0.000, z=-8.576, rx=-0.000, ry=0.000, rz=-0.000, shoulder=lefty, elbow=epositive, wrist=wpositive, fatherId=fReference[0]}
  [1080] = {x=-21.420, y=0.000, z=-8.585, rx=-0.000, ry=0.000, rz=-0.000, shoulder=lefty, elbow=epositive, wrist=wpositive, fatherId=fReference[0]}
  [1081] = {x=-20.914, y=0.000, z=-8.594, rx=-0.000, ry=0.000, rz=-0.000, shoulder=lefty, elbow=epositive, wrist=wpositive, fatherId=fReference[0]}
  [1082] = {x=-20.407, y=0.000, z=-8.602, rx=-0.000, ry=0.000, rz=-0.000, shoulder=lefty, elbow=epositive, wrist=wpositive, fatherId=fReference[0]}
  [1083] = {x=-19.899, y=0.000, z=-8.611, rx=-0.000, ry=0.000, rz=-0.000, shoulder=lefty, elbow=epositive, wrist=wpositive, fatherId=fReference[0]}
  [1084] = {x=-19.390, y=0.000, z=-8.621, rx=-0.000, ry=0.000, rz=-0.000, shoulder=lefty, elbow=epositive, wrist=wpositive, fatherId=fReference[0]}
  [1085] = {x=-18.883, y=0.000, z=-8.630, rx=-0.000, ry=0.000, rz=-0.000, shoulder=lefty, elbow=epositive, wrist=wpositive, fatherId=fReference[0]}
  [1086] = {x=-18.376, y=0.000, z=-8.639, rx=-0.000, ry=0.000, rz=-0.000, shoulder=lefty, elbow=epositive, wrist=wpositive, fatherId=fReference[0]}
  [1087] = {x=-17.868, y=0.000, z=-8.649, rx=-0.000, ry=0.000, rz=-0.000, shoulder=lefty, elbow=epositive, wrist=wpositive, fatherId=fReference[0]}
  [1088] = {x=-17.360, y=0.000, z=-8.658, rx=-0.000, ry=0.000, rz=-0.000, shoulder=lefty, elbow=epositive, wrist=wpositive, fatherId=fReference[0]}
  [1089] = {x=-16.852, y=0.000, z=-8.668, rx=-0.000, ry=0.000, rz=-0.000, shoulder=lefty, elbow=epositive, wrist=wpositive, fatherId=fReference[0]}
  [1090] = {x=-16.343, y=0.000, z=-8.677, rx=-0.000, ry=0.000, rz=-0.000, shoulder=lefty, elbow=epositive, wrist=wpositive, fatherId=fReference[0]}
  [1091] = {x=-15.835, y=0.000, z=-8.687, rx=-0.000, ry=0.000, rz=-0.000, shoulder=lefty, elbow=epositive, wrist=wpositive, fatherId=fReference[0]}
  [1092] = {x=-15.325, y=0.000, z=-8.696, rx=-0.000, ry=0.000, rz=-0.000, shoulder=lefty, elbow=epositive, wrist=wpositive, fatherId=fReference[0]}
  [1093] = {x=-14.816, y=0.000, z=-8.706, rx=-0.000, ry=0.000, rz=-0.000, shoulder=lefty, elbow=epositive, wrist=wpositive, fatherId=fReference[0]}
  [1094] = {x=-14.309, y=0.000, z=-8.715, rx=-0.000, ry=0.000, rz=-0.000, shoulder=lefty, elbow=epositive, wrist=wpositive, fatherId=fReference[0]}
  [1095] = {x=-13.802, y=0.000, z=-8.724, rx=-0.000, ry=0.000, rz=-0.000, shoulder=lefty, elbow=epositive, wrist=wpositive, fatherId=fReference[0]}
  [1096] = {x=-13.297, y=0.000, z=-8.733, rx=-0.000, ry=0.000, rz=-0.000, shoulder=lefty, elbow=epositive, wrist=wpositive, fatherId=fReference[0]}
  [1097] = {x=-12.792, y=0.000, z=-8.742, rx=-0.000, ry=0.000, rz=-0.000, shoulder=lefty, elbow=epositive, wrist=wpositive, fatherId=fReference[0]}
  [1098] = {x=-12.287, y=0.000, z=-8.750, rx=-0.000, ry=0.000, rz=-0.000, shoulder=lefty, elbow=epositive, wrist=wpositive, fatherId=fReference[0]}
  [1099] = {x=-11.783, y=0.000, z=-8.758, rx=-0.000, ry=0.000, rz=-0.000, shoulder=lefty, elbow=epositive, wrist=wpositive, fatherId=fReference[0]}
  [1100] = {x=-11.278, y=0.000, z=-8.766, rx=-0.000, ry=0.000, rz=-0.000, shoulder=lefty, elbow=epositive, wrist=wpositive, fatherId=fReference[0]}
  [1101] = {x=-10.774, y=0.000, z=-8.774, rx=-0.000, ry=0.000, rz=-0.000, shoulder=lefty, elbow=epositive, wrist=wpositive, fatherId=fReference[0]}
  [1102] = {x=-10.270, y=0.000, z=-8.783, rx=-0.000, ry=0.000, rz=-0.000, shoulder=lefty, elbow=epositive, wrist=wpositive, fatherId=fReference[0]}
  [1103] = {x=-9.764, y=0.000, z=-8.791, rx=-0.000, ry=0.000, rz=-0.000, shoulder=lefty, elbow=epositive, wrist=wpositive, fatherId=fReference[0]}
  [1104] = {x=-9.260, y=0.000, z=-8.800, rx=-0.000, ry=0.000, rz=-0.000, shoulder=lefty, elbow=epositive, wrist=wpositive, fatherId=fReference[0]}
  [1105] = {x=-8.754, y=0.000, z=-8.808, rx=-0.000, ry=0.000, rz=-0.000, shoulder=lefty, elbow=epositive, wrist=wpositive, fatherId=fReference[0]}
  [1106] = {x=-8.249, y=0.000, z=-8.816, rx=-0.000, ry=0.000, rz=-0.000, shoulder=lefty, elbow=epositive, wrist=wpositive, fatherId=fReference[0]}
  [1107] = {x=-7.745, y=0.000, z=-8.825, rx=-0.000, ry=0.000, rz=-0.000, shoulder=lefty, elbow=epositive, wrist=wpositive, fatherId=fReference[0]}
  [1108] = {x=-7.239, y=0.000, z=-8.833, rx=-0.000, ry=0.000, rz=-0.000, shoulder=lefty, elbow=epositive, wrist=wpositive, fatherId=fReference[0]}
  [1109] = {x=-6.735, y=0.000, z=-8.842, rx=-0.000, ry=0.000, rz=-0.000, shoulder=lefty, elbow=epositive, wrist=wpositive, fatherId=fReference[0]}
  [1110] = {x=-6.229, y=0.000, z=-8.850, rx=-0.000, ry=0.000, rz=-0.000, shoulder=lefty, elbow=epositive, wrist=wpositive, fatherId=fReference[0]}
  [1111] = {x=-5.725, y=0.000, z=-8.858, rx=-0.000, ry=0.000, rz=-0.000, shoulder=lefty, elbow=epositive, wrist=wpositive, fatherId=fReference[0]}
  [1112] = {x=-5.218, y=0.000, z=-8.866, rx=-0.000, ry=0.000, rz=-0.000, shoulder=lefty, elbow=epositive, wrist=wpositive, fatherId=fReference[0]}
  [1113] = {x=-4.713, y=0.000, z=-8.874, rx=-0.000, ry=0.000, rz=-0.000, shoulder=lefty, elbow=epositive, wrist=wpositive, fatherId=fReference[0]}
  [1114] = {x=-4.208, y=0.000, z=-8.882, rx=-0.000, ry=0.000, rz=-0.000, shoulder=lefty, elbow=epositive, wrist=wpositive, fatherId=fReference[0]}
  [1115] = {x=-3.704, y=0.000, z=-8.890, rx=-0.000, ry=0.000, rz=-0.000, shoulder=lefty, elbow=epositive, wrist=wpositive, fatherId=fReference[0]}
  [1116] = {x=-3.197, y=0.000, z=-8.898, rx=-0.000, ry=0.000, rz=-0.000, shoulder=lefty, elbow=epositive, wrist=wpositive, fatherId=fReference[0]}
  [1117] = {x=-2.689, y=0.000, z=-8.907, rx=-0.000, ry=0.000, rz=-0.000, shoulder=lefty, elbow=epositive, wrist=wpositive, fatherId=fReference[0]}
  [1118] = {x=-2.181, y=0.000, z=-8.915, rx=-0.000, ry=0.000, rz=-0.000, shoulder=lefty, elbow=epositive, wrist=wpositive, fatherId=fReference[0]}
  [1119] = {x=-1.674, y=0.000, z=-8.924, rx=-0.000, ry=0.000, rz=-0.000, shoulder=lefty, elbow=epositive, wrist=wpositive, fatherId=fReference[0]}
  [1120] = {x=-1.165, y=0.000, z=-8.931, rx=-0.000, ry=0.000, rz=-0.000, shoulder=lefty, elbow=epositive, wrist=wpositive, fatherId=fReference[0]}
  [1121] = {x=-0.654, y=0.000, z=-8.939, rx=-0.000, ry=0.000, rz=-0.000, shoulder=lefty, elbow=epositive, wrist=wpositive, fatherId=fReference[0]}
  [1122] = {x=-0.144, y=0.000, z=-8.947, rx=-0.000, ry=0.000, rz=-0.000, shoulder=lefty, elbow=epositive, wrist=wpositive, fatherId=fReference[0]}
  [1123] = {x=0.365, y=0.000, z=-8.956, rx=-0.000, ry=0.000, rz=-0.000, shoulder=lefty, elbow=epositive, wrist=wpositive, fatherId=fReference[0]}
  [1124] = {x=0.876, y=0.000, z=-8.964, rx=-0.000, ry=0.000, rz=-0.000, shoulder=lefty, elbow=epositive, wrist=wpositive, fatherId=fReference[0]}
  [1125] = {x=1.386, y=0.000, z=-8.972, rx=-0.000, ry=0.000, rz=-0.000, shoulder=lefty, elbow=epositive, wrist=wpositive, fatherId=fReference[0]}
  [1126] = {x=1.898, y=0.000, z=-8.981, rx=-0.000, ry=0.000, rz=-0.000, shoulder=lefty, elbow=epositive, wrist=wpositive, fatherId=fReference[0]}
  [1127] = {x=2.409, y=0.000, z=-8.989, rx=-0.000, ry=0.000, rz=-0.000, shoulder=lefty, elbow=epositive, wrist=wpositive, fatherId=fReference[0]}
  [1128] = {x=2.919, y=0.000, z=-8.998, rx=-0.000, ry=0.000, rz=-0.000, shoulder=lefty, elbow=epositive, wrist=wpositive, fatherId=fReference[0]}
  [1129] = {x=3.430, y=0.000, z=-9.006, rx=-0.000, ry=0.000, rz=-0.000, shoulder=lefty, elbow=epositive, wrist=wpositive, fatherId=fReference[0]}
  [1130] = {x=3.938, y=0.000, z=-9.015, rx=-0.000, ry=0.000, rz=-0.000, shoulder=lefty, elbow=epositive, wrist=wpositive, fatherId=fReference[0]}
  [1131] = {x=4.448, y=0.000, z=-9.024, rx=-0.000, ry=0.000, rz=-0.000, shoulder=lefty, elbow=epositive, wrist=wpositive, fatherId=fReference[0]}
  [1132] = {x=4.958, y=0.000, z=-9.033, rx=-0.000, ry=0.000, rz=-0.000, shoulder=lefty, elbow=epositive, wrist=wpositive, fatherId=fReference[0]}
  [1133] = {x=5.467, y=0.000, z=-9.042, rx=-0.000, ry=0.000, rz=-0.000, shoulder=lefty, elbow=epositive, wrist=wpositive, fatherId=fReference[0]}
  [1134] = {x=5.976, y=0.000, z=-9.050, rx=-0.000, ry=0.000, rz=-0.000, shoulder=lefty, elbow=epositive, wrist=wpositive, fatherId=fReference[0]}
  [1135] = {x=6.486, y=0.000, z=-9.059, rx=-0.000, ry=0.000, rz=-0.000, shoulder=lefty, elbow=epositive, wrist=wpositive, fatherId=fReference[0]}
  [1136] = {x=6.994, y=0.000, z=-9.068, rx=-0.000, ry=0.000, rz=-0.000, shoulder=lefty, elbow=epositive, wrist=wpositive, fatherId=fReference[0]}
  [1137] = {x=7.503, y=0.000, z=-9.077, rx=-0.000, ry=0.000, rz=-0.000, shoulder=lefty, elbow=epositive, wrist=wpositive, fatherId=fReference[0]}
  [1138] = {x=8.010, y=0.000, z=-9.086, rx=-0.000, ry=0.000, rz=-0.000, shoulder=lefty, elbow=epositive, wrist=wpositive, fatherId=fReference[0]}
  [1139] = {x=8.517, y=0.000, z=-9.096, rx=-0.000, ry=0.000, rz=-0.000, shoulder=lefty, elbow=epositive, wrist=wpositive, fatherId=fReference[0]}
  [1140] = {x=9.027, y=0.000, z=-9.104, rx=-0.000, ry=0.000, rz=-0.000, shoulder=lefty, elbow=epositive, wrist=wpositive, fatherId=fReference[0]}
  [1141] = {x=9.536, y=0.000, z=-9.114, rx=-0.000, ry=0.000, rz=-0.000, shoulder=lefty, elbow=epositive, wrist=wpositive, fatherId=fReference[0]}
  [1142] = {x=10.045, y=0.000, z=-9.123, rx=-0.000, ry=0.000, rz=-0.000, shoulder=lefty, elbow=epositive, wrist=wpositive, fatherId=fReference[0]}
  [1143] = {x=10.553, y=0.000, z=-9.131, rx=-0.000, ry=0.000, rz=-0.000, shoulder=lefty, elbow=epositive, wrist=wpositive, fatherId=fReference[0]}
  [1144] = {x=11.061, y=0.000, z=-9.139, rx=-0.000, ry=0.000, rz=-0.000, shoulder=lefty, elbow=epositive, wrist=wpositive, fatherId=fReference[0]}
  [1145] = {x=11.570, y=0.000, z=-9.150, rx=-0.000, ry=0.000, rz=-0.000, shoulder=lefty, elbow=epositive, wrist=wpositive, fatherId=fReference[0]}
  [1146] = {x=12.079, y=0.000, z=-9.159, rx=-0.000, ry=0.000, rz=-0.000, shoulder=lefty, elbow=epositive, wrist=wpositive, fatherId=fReference[0]}
  [1147] = {x=12.587, y=0.000, z=-9.168, rx=-0.000, ry=0.000, rz=-0.000, shoulder=lefty, elbow=epositive, wrist=wpositive, fatherId=fReference[0]}
  [1148] = {x=13.096, y=0.000, z=-9.177, rx=-0.000, ry=0.000, rz=-0.000, shoulder=lefty, elbow=epositive, wrist=wpositive, fatherId=fReference[0]}
  [1149] = {x=13.605, y=0.000, z=-9.187, rx=-0.000, ry=0.000, rz=-0.000, shoulder=lefty, elbow=epositive, wrist=wpositive, fatherId=fReference[0]}
  [1150] = {x=14.114, y=0.000, z=-9.196, rx=-0.000, ry=0.000, rz=-0.000, shoulder=lefty, elbow=epositive, wrist=wpositive, fatherId=fReference[0]}
  [1151] = {x=14.624, y=0.000, z=-9.206, rx=-0.000, ry=0.000, rz=-0.000, shoulder=lefty, elbow=epositive, wrist=wpositive, fatherId=fReference[0]}
  [1152] = {x=15.135, y=0.000, z=-9.215, rx=-0.000, ry=0.000, rz=-0.000, shoulder=lefty, elbow=epositive, wrist=wpositive, fatherId=fReference[0]}
  [1153] = {x=15.646, y=0.000, z=-9.224, rx=-0.000, ry=0.000, rz=-0.000, shoulder=lefty, elbow=epositive, wrist=wpositive, fatherId=fReference[0]}
  [1154] = {x=16.157, y=0.000, z=-9.234, rx=-0.000, ry=0.000, rz=-0.000, shoulder=lefty, elbow=epositive, wrist=wpositive, fatherId=fReference[0]}
  [1155] = {x=16.666, y=0.000, z=-9.243, rx=-0.000, ry=0.000, rz=-0.000, shoulder=lefty, elbow=epositive, wrist=wpositive, fatherId=fReference[0]}
  [1156] = {x=17.178, y=0.000, z=-9.253, rx=-0.000, ry=0.000, rz=-0.000, shoulder=lefty, elbow=epositive, wrist=wpositive, fatherId=fReference[0]}
  [1157] = {x=17.691, y=0.000, z=-9.262, rx=-0.000, ry=0.000, rz=-0.000, shoulder=lefty, elbow=epositive, wrist=wpositive, fatherId=fReference[0]}
  [1158] = {x=18.201, y=0.000, z=-9.271, rx=-0.000, ry=0.000, rz=-0.000, shoulder=lefty, elbow=epositive, wrist=wpositive, fatherId=fReference[0]}
  [1159] = {x=18.714, y=0.000, z=-9.281, rx=-0.000, ry=0.000, rz=-0.000, shoulder=lefty, elbow=epositive, wrist=wpositive, fatherId=fReference[0]}
  [1160] = {x=19.227, y=0.000, z=-9.291, rx=-0.000, ry=0.000, rz=-0.000, shoulder=lefty, elbow=epositive, wrist=wpositive, fatherId=fReference[0]}
  [1161] = {x=19.742, y=0.000, z=-9.299, rx=-0.000, ry=0.000, rz=-0.000, shoulder=lefty, elbow=epositive, wrist=wpositive, fatherId=fReference[0]}
  [1162] = {x=20.257, y=0.000, z=-9.309, rx=-0.000, ry=0.000, rz=-0.000, shoulder=lefty, elbow=epositive, wrist=wpositive, fatherId=fReference[0]}
  [1163] = {x=20.772, y=0.000, z=-9.319, rx=-0.000, ry=0.000, rz=-0.000, shoulder=lefty, elbow=epositive, wrist=wpositive, fatherId=fReference[0]}
  [1164] = {x=21.288, y=0.000, z=-9.328, rx=-0.000, ry=0.000, rz=-0.000, shoulder=lefty, elbow=epositive, wrist=wpositive, fatherId=fReference[0]}
  [1165] = {x=21.805, y=0.000, z=-9.338, rx=-0.000, ry=0.000, rz=-0.000, shoulder=lefty, elbow=epositive, wrist=wpositive, fatherId=fReference[0]}
  [1166] = {x=22.322, y=0.000, z=-9.348, rx=-0.000, ry=0.000, rz=-0.000, shoulder=lefty, elbow=epositive, wrist=wpositive, fatherId=fReference[0]}
  [1167] = {x=22.838, y=0.000, z=-9.357, rx=-0.000, ry=0.000, rz=-0.000, shoulder=lefty, elbow=epositive, wrist=wpositive, fatherId=fReference[0]}
  [1168] = {x=23.356, y=0.000, z=-9.368, rx=-0.000, ry=0.000, rz=-0.000, shoulder=lefty, elbow=epositive, wrist=wpositive, fatherId=fReference[0]}
  [1169] = {x=23.877, y=0.000, z=-9.380, rx=-0.000, ry=0.000, rz=-0.000, shoulder=lefty, elbow=epositive, wrist=wpositive, fatherId=fReference[0]}
  [1170] = {x=24.398, y=0.000, z=-9.389, rx=-0.000, ry=0.000, rz=-0.000, shoulder=lefty, elbow=epositive, wrist=wpositive, fatherId=fReference[0]}
  [1171] = {x=24.915, y=0.000, z=-9.399, rx=-0.000, ry=0.000, rz=-0.000, shoulder=lefty, elbow=epositive, wrist=wpositive, fatherId=fReference[0]}
  [1172] = {x=25.441, y=0.000, z=-9.409, rx=-0.000, ry=0.000, rz=-0.000, shoulder=lefty, elbow=epositive, wrist=wpositive, fatherId=fReference[0]}
  [1173] = {x=25.964, y=0.000, z=-9.421, rx=-0.000, ry=0.000, rz=-0.000, shoulder=lefty, elbow=epositive, wrist=wpositive, fatherId=fReference[0]}
  [1174] = {x=26.489, y=0.000, z=-9.434, rx=-0.000, ry=0.000, rz=-0.000, shoulder=lefty, elbow=epositive, wrist=wpositive, fatherId=fReference[0]}
  [1175] = {x=27.016, y=0.000, z=-9.446, rx=-0.000, ry=0.000, rz=-0.000, shoulder=lefty, elbow=epositive, wrist=wpositive, fatherId=fReference[0]}
  [1176] = {x=27.545, y=0.000, z=-9.460, rx=-0.000, ry=0.000, rz=-0.000, shoulder=lefty, elbow=epositive, wrist=wpositive, fatherId=fReference[0]}
  [1177] = {x=28.078, y=0.000, z=-9.474, rx=-0.000, ry=0.000, rz=-0.000, shoulder=lefty, elbow=epositive, wrist=wpositive, fatherId=fReference[0]}
  [1178] = {x=28.613, y=0.000, z=-9.487, rx=-0.000, ry=0.000, rz=-0.000, shoulder=lefty, elbow=epositive, wrist=wpositive, fatherId=fReference[0]}
  [1179] = {x=29.147, y=0.000, z=-9.502, rx=-0.000, ry=0.000, rz=-0.000, shoulder=lefty, elbow=epositive, wrist=wpositive, fatherId=fReference[0]}
  [1180] = {x=29.691, y=0.000, z=-9.518, rx=-0.000, ry=0.000, rz=-0.000, shoulder=lefty, elbow=epositive, wrist=wpositive, fatherId=fReference[0]}
  [1181] = {x=30.234, y=0.000, z=-9.532, rx=-0.000, ry=0.000, rz=-0.000, shoulder=lefty, elbow=epositive, wrist=wpositive, fatherId=fReference[0]}
  [1182] = {x=30.783, y=0.000, z=-9.548, rx=-0.000, ry=0.000, rz=-0.000, shoulder=lefty, elbow=epositive, wrist=wpositive, fatherId=fReference[0]}
  [1183] = {x=31.344, y=0.000, z=-9.564, rx=-0.000, ry=0.000, rz=-0.000, shoulder=lefty, elbow=epositive, wrist=wpositive, fatherId=fReference[0]}
  [1184] = {x=31.916, y=0.000, z=-9.582, rx=-0.000, ry=0.000, rz=-0.000, shoulder=lefty, elbow=epositive, wrist=wpositive, fatherId=fReference[0]}
  [1185] = {x=32.507, y=0.000, z=-9.598, rx=-0.000, ry=0.000, rz=-0.000, shoulder=lefty, elbow=epositive, wrist=wpositive, fatherId=fReference[0]}
  [1186] = {x=33.112, y=0.000, z=-9.614, rx=-0.000, ry=0.000, rz=-0.000, shoulder=lefty, elbow=epositive, wrist=wpositive, fatherId=fReference[0]}
  [1187] = {x=33.718, y=0.000, z=-9.626, rx=-0.000, ry=0.000, rz=-0.000, shoulder=lefty, elbow=epositive, wrist=wpositive, fatherId=fReference[0]}
  [1188] = {x=34.293, y=0.000, z=-9.634, rx=-0.000, ry=0.000, rz=-0.000, shoulder=lefty, elbow=epositive, wrist=wpositive, fatherId=fReference[0]}
  [1189] = {x=32.555, y=0.000, z=-9.653, rx=-0.000, ry=0.000, rz=-0.000, shoulder=lefty, elbow=epositive, wrist=wpositive, fatherId=fReference[0]}
  [1190] = {x=31.771, y=0.000, z=-9.624, rx=-0.000, ry=0.000, rz=-0.000, shoulder=lefty, elbow=epositive, wrist=wpositive, fatherId=fReference[0]}
  [1191] = {x=31.152, y=0.000, z=-9.608, rx=-0.000, ry=0.000, rz=-0.000, shoulder=lefty, elbow=epositive, wrist=wpositive, fatherId=fReference[0]}
  [1192] = {x=30.567, y=0.000, z=-9.598, rx=-0.000, ry=0.000, rz=-0.000, shoulder=lefty, elbow=epositive, wrist=wpositive, fatherId=fReference[0]}
  [1193] = {x=30.003, y=0.000, z=-9.592, rx=-0.000, ry=0.000, rz=-0.000, shoulder=lefty, elbow=epositive, wrist=wpositive, fatherId=fReference[0]}
  [1194] = {x=29.456, y=0.000, z=-9.589, rx=-0.000, ry=0.000, rz=-0.000, shoulder=lefty, elbow=epositive, wrist=wpositive, fatherId=fReference[0]}
  [1195] = {x=28.917, y=0.000, z=-9.588, rx=-0.000, ry=0.000, rz=-0.000, shoulder=lefty, elbow=epositive, wrist=wpositive, fatherId=fReference[0]}
  [1196] = {x=28.385, y=0.000, z=-9.590, rx=-0.000, ry=0.000, rz=-0.000, shoulder=lefty, elbow=epositive, wrist=wpositive, fatherId=fReference[0]}
  [1197] = {x=27.860, y=0.000, z=-9.592, rx=-0.000, ry=0.000, rz=-0.000, shoulder=lefty, elbow=epositive, wrist=wpositive, fatherId=fReference[0]}
  [1198] = {x=27.339, y=0.000, z=-9.597, rx=-0.000, ry=0.000, rz=-0.000, shoulder=lefty, elbow=epositive, wrist=wpositive, fatherId=fReference[0]}
  [1199] = {x=26.823, y=0.000, z=-9.602, rx=-0.000, ry=0.000, rz=-0.000, shoulder=lefty, elbow=epositive, wrist=wpositive, fatherId=fReference[0]}
  [1200] = {x=26.309, y=0.000, z=-9.608, rx=-0.000, ry=0.000, rz=-0.000, shoulder=lefty, elbow=epositive, wrist=wpositive, fatherId=fReference[0]}
  [1201] = {x=25.801, y=0.000, z=-9.616, rx=-0.000, ry=0.000, rz=-0.000, shoulder=lefty, elbow=epositive, wrist=wpositive, fatherId=fReference[0]}
  [1202] = {x=25.293, y=0.000, z=-9.625, rx=-0.000, ry=0.000, rz=-0.000, shoulder=lefty, elbow=epositive, wrist=wpositive, fatherId=fReference[0]}
  [1203] = {x=24.788, y=0.000, z=-9.634, rx=-0.000, ry=0.000, rz=-0.000, shoulder=lefty, elbow=epositive, wrist=wpositive, fatherId=fReference[0]}
  [1204] = {x=24.289, y=0.000, z=-9.645, rx=-0.000, ry=0.000, rz=-0.000, shoulder=lefty, elbow=epositive, wrist=wpositive, fatherId=fReference[0]}
  [1205] = {x=23.792, y=0.000, z=-9.655, rx=-0.000, ry=0.000, rz=-0.000, shoulder=lefty, elbow=epositive, wrist=wpositive, fatherId=fReference[0]}
  [1206] = {x=23.293, y=0.000, z=-9.665, rx=-0.000, ry=0.000, rz=-0.000, shoulder=lefty, elbow=epositive, wrist=wpositive, fatherId=fReference[0]}
  [1207] = {x=22.795, y=0.000, z=-9.676, rx=-0.000, ry=0.000, rz=-0.000, shoulder=lefty, elbow=epositive, wrist=wpositive, fatherId=fReference[0]}
  [1208] = {x=22.298, y=0.000, z=-9.687, rx=-0.000, ry=0.000, rz=-0.000, shoulder=lefty, elbow=epositive, wrist=wpositive, fatherId=fReference[0]}
  [1209] = {x=21.803, y=0.000, z=-9.698, rx=-0.000, ry=0.000, rz=-0.000, shoulder=lefty, elbow=epositive, wrist=wpositive, fatherId=fReference[0]}
  [1210] = {x=21.307, y=0.000, z=-9.709, rx=-0.000, ry=0.000, rz=-0.000, shoulder=lefty, elbow=epositive, wrist=wpositive, fatherId=fReference[0]}
  [1211] = {x=20.811, y=0.000, z=-9.720, rx=-0.000, ry=0.000, rz=-0.000, shoulder=lefty, elbow=epositive, wrist=wpositive, fatherId=fReference[0]}
  [1212] = {x=20.313, y=0.000, z=-9.730, rx=-0.000, ry=0.000, rz=-0.000, shoulder=lefty, elbow=epositive, wrist=wpositive, fatherId=fReference[0]}
  [1213] = {x=19.815, y=0.000, z=-9.741, rx=-0.000, ry=0.000, rz=-0.000, shoulder=lefty, elbow=epositive, wrist=wpositive, fatherId=fReference[0]}
  [1214] = {x=19.318, y=0.000, z=-9.751, rx=-0.000, ry=0.000, rz=-0.000, shoulder=lefty, elbow=epositive, wrist=wpositive, fatherId=fReference[0]}
  [1215] = {x=18.820, y=0.000, z=-9.761, rx=-0.000, ry=0.000, rz=-0.000, shoulder=lefty, elbow=epositive, wrist=wpositive, fatherId=fReference[0]}
  [1216] = {x=18.321, y=0.000, z=-9.771, rx=-0.000, ry=0.000, rz=-0.000, shoulder=lefty, elbow=epositive, wrist=wpositive, fatherId=fReference[0]}
  [1217] = {x=17.823, y=0.000, z=-9.781, rx=-0.000, ry=0.000, rz=-0.000, shoulder=lefty, elbow=epositive, wrist=wpositive, fatherId=fReference[0]}
  [1218] = {x=17.324, y=0.000, z=-9.791, rx=-0.000, ry=0.000, rz=-0.000, shoulder=lefty, elbow=epositive, wrist=wpositive, fatherId=fReference[0]}
  [1219] = {x=16.824, y=0.000, z=-9.801, rx=-0.000, ry=0.000, rz=-0.000, shoulder=lefty, elbow=epositive, wrist=wpositive, fatherId=fReference[0]}
  [1220] = {x=16.323, y=0.000, z=-9.810, rx=-0.000, ry=0.000, rz=-0.000, shoulder=lefty, elbow=epositive, wrist=wpositive, fatherId=fReference[0]}
  [1221] = {x=15.823, y=0.000, z=-9.820, rx=-0.000, ry=0.000, rz=-0.000, shoulder=lefty, elbow=epositive, wrist=wpositive, fatherId=fReference[0]}
  [1222] = {x=15.322, y=0.000, z=-9.829, rx=-0.000, ry=0.000, rz=-0.000, shoulder=lefty, elbow=epositive, wrist=wpositive, fatherId=fReference[0]}
  [1223] = {x=14.821, y=0.000, z=-9.838, rx=-0.000, ry=0.000, rz=-0.000, shoulder=lefty, elbow=epositive, wrist=wpositive, fatherId=fReference[0]}
  [1224] = {x=14.320, y=0.000, z=-9.847, rx=-0.000, ry=0.000, rz=-0.000, shoulder=lefty, elbow=epositive, wrist=wpositive, fatherId=fReference[0]}
  [1225] = {x=13.818, y=0.000, z=-9.856, rx=-0.000, ry=0.000, rz=-0.000, shoulder=lefty, elbow=epositive, wrist=wpositive, fatherId=fReference[0]}
  [1226] = {x=13.315, y=0.000, z=-9.866, rx=-0.000, ry=0.000, rz=-0.000, shoulder=lefty, elbow=epositive, wrist=wpositive, fatherId=fReference[0]}
  [1227] = {x=12.813, y=0.000, z=-9.875, rx=-0.000, ry=0.000, rz=-0.000, shoulder=lefty, elbow=epositive, wrist=wpositive, fatherId=fReference[0]}
  [1228] = {x=12.311, y=0.000, z=-9.884, rx=-0.000, ry=0.000, rz=-0.000, shoulder=lefty, elbow=epositive, wrist=wpositive, fatherId=fReference[0]}
  [1229] = {x=11.809, y=0.000, z=-9.893, rx=-0.000, ry=0.000, rz=-0.000, shoulder=lefty, elbow=epositive, wrist=wpositive, fatherId=fReference[0]}
  [1230] = {x=11.305, y=0.000, z=-9.902, rx=-0.000, ry=0.000, rz=-0.000, shoulder=lefty, elbow=epositive, wrist=wpositive, fatherId=fReference[0]}
  [1231] = {x=10.801, y=0.000, z=-9.911, rx=-0.000, ry=0.000, rz=-0.000, shoulder=lefty, elbow=epositive, wrist=wpositive, fatherId=fReference[0]}
  [1232] = {x=10.297, y=0.000, z=-9.920, rx=-0.000, ry=0.000, rz=-0.000, shoulder=lefty, elbow=epositive, wrist=wpositive, fatherId=fReference[0]}
  [1233] = {x=9.795, y=0.000, z=-9.930, rx=-0.000, ry=0.000, rz=-0.000, shoulder=lefty, elbow=epositive, wrist=wpositive, fatherId=fReference[0]}
  [1234] = {x=9.293, y=0.000, z=-9.939, rx=-0.000, ry=0.000, rz=-0.000, shoulder=lefty, elbow=epositive, wrist=wpositive, fatherId=fReference[0]}
  [1235] = {x=8.791, y=0.000, z=-9.948, rx=-0.000, ry=0.000, rz=-0.000, shoulder=lefty, elbow=epositive, wrist=wpositive, fatherId=fReference[0]}
  [1236] = {x=8.287, y=0.000, z=-9.957, rx=-0.000, ry=0.000, rz=-0.000, shoulder=lefty, elbow=epositive, wrist=wpositive, fatherId=fReference[0]}
  [1237] = {x=7.784, y=0.000, z=-9.967, rx=-0.000, ry=0.000, rz=-0.000, shoulder=lefty, elbow=epositive, wrist=wpositive, fatherId=fReference[0]}
  [1238] = {x=7.281, y=0.000, z=-9.976, rx=-0.000, ry=0.000, rz=-0.000, shoulder=lefty, elbow=epositive, wrist=wpositive, fatherId=fReference[0]}
  [1239] = {x=6.779, y=0.000, z=-9.986, rx=-0.000, ry=0.000, rz=-0.000, shoulder=lefty, elbow=epositive, wrist=wpositive, fatherId=fReference[0]}
  [1240] = {x=6.277, y=0.000, z=-9.996, rx=-0.000, ry=0.000, rz=-0.000, shoulder=lefty, elbow=epositive, wrist=wpositive, fatherId=fReference[0]}
  [1241] = {x=5.774, y=0.000, z=-10.006, rx=-0.000, ry=0.000, rz=-0.000, shoulder=lefty, elbow=epositive, wrist=wpositive, fatherId=fReference[0]}
  [1242] = {x=5.271, y=0.000, z=-10.016, rx=-0.000, ry=0.000, rz=-0.000, shoulder=lefty, elbow=epositive, wrist=wpositive, fatherId=fReference[0]}
  [1243] = {x=4.769, y=0.000, z=-10.026, rx=-0.000, ry=0.000, rz=-0.000, shoulder=lefty, elbow=epositive, wrist=wpositive, fatherId=fReference[0]}
  [1244] = {x=4.267, y=0.000, z=-10.036, rx=-0.000, ry=0.000, rz=-0.000, shoulder=lefty, elbow=epositive, wrist=wpositive, fatherId=fReference[0]}
  [1245] = {x=3.764, y=0.000, z=-10.046, rx=-0.000, ry=0.000, rz=-0.000, shoulder=lefty, elbow=epositive, wrist=wpositive, fatherId=fReference[0]}
  [1246] = {x=3.260, y=0.000, z=-10.057, rx=-0.000, ry=0.000, rz=-0.000, shoulder=lefty, elbow=epositive, wrist=wpositive, fatherId=fReference[0]}
  [1247] = {x=2.757, y=0.000, z=-10.067, rx=-0.000, ry=0.000, rz=-0.000, shoulder=lefty, elbow=epositive, wrist=wpositive, fatherId=fReference[0]}
  [1248] = {x=2.255, y=0.000, z=-10.078, rx=-0.000, ry=0.000, rz=-0.000, shoulder=lefty, elbow=epositive, wrist=wpositive, fatherId=fReference[0]}
  [1249] = {x=1.752, y=0.000, z=-10.088, rx=-0.000, ry=0.000, rz=-0.000, shoulder=lefty, elbow=epositive, wrist=wpositive, fatherId=fReference[0]}
  [1250] = {x=1.251, y=0.000, z=-10.098, rx=-0.000, ry=0.000, rz=-0.000, shoulder=lefty, elbow=epositive, wrist=wpositive, fatherId=fReference[0]}
  [1251] = {x=0.749, y=0.000, z=-10.109, rx=-0.000, ry=0.000, rz=-0.000, shoulder=lefty, elbow=epositive, wrist=wpositive, fatherId=fReference[0]}
  [1252] = {x=0.247, y=0.000, z=-10.119, rx=-0.000, ry=0.000, rz=-0.000, shoulder=lefty, elbow=epositive, wrist=wpositive, fatherId=fReference[0]}
  [1253] = {x=-0.255, y=0.000, z=-10.129, rx=-0.000, ry=0.000, rz=-0.000, shoulder=lefty, elbow=epositive, wrist=wpositive, fatherId=fReference[0]}
  [1254] = {x=-0.757, y=0.000, z=-10.139, rx=-0.000, ry=0.000, rz=-0.000, shoulder=lefty, elbow=epositive, wrist=wpositive, fatherId=fReference[0]}
  [1255] = {x=-1.260, y=0.000, z=-10.149, rx=-0.000, ry=0.000, rz=-0.000, shoulder=lefty, elbow=epositive, wrist=wpositive, fatherId=fReference[0]}
  [1256] = {x=-1.761, y=0.000, z=-10.159, rx=-0.000, ry=0.000, rz=-0.000, shoulder=lefty, elbow=epositive, wrist=wpositive, fatherId=fReference[0]}
  [1257] = {x=-2.262, y=0.000, z=-10.169, rx=-0.000, ry=0.000, rz=-0.000, shoulder=lefty, elbow=epositive, wrist=wpositive, fatherId=fReference[0]}
  [1258] = {x=-2.764, y=0.000, z=-10.178, rx=-0.000, ry=0.000, rz=-0.000, shoulder=lefty, elbow=epositive, wrist=wpositive, fatherId=fReference[0]}
  [1259] = {x=-3.265, y=0.000, z=-10.188, rx=-0.000, ry=0.000, rz=-0.000, shoulder=lefty, elbow=epositive, wrist=wpositive, fatherId=fReference[0]}
  [1260] = {x=-3.767, y=0.000, z=-10.198, rx=-0.000, ry=0.000, rz=-0.000, shoulder=lefty, elbow=epositive, wrist=wpositive, fatherId=fReference[0]}
  [1261] = {x=-4.268, y=0.000, z=-10.208, rx=-0.000, ry=0.000, rz=-0.000, shoulder=lefty, elbow=epositive, wrist=wpositive, fatherId=fReference[0]}
  [1262] = {x=-4.771, y=0.000, z=-10.218, rx=-0.000, ry=0.000, rz=-0.000, shoulder=lefty, elbow=epositive, wrist=wpositive, fatherId=fReference[0]}
  [1263] = {x=-5.273, y=0.000, z=-10.227, rx=-0.000, ry=0.000, rz=-0.000, shoulder=lefty, elbow=epositive, wrist=wpositive, fatherId=fReference[0]}
  [1264] = {x=-5.775, y=0.000, z=-10.237, rx=-0.000, ry=0.000, rz=-0.000, shoulder=lefty, elbow=epositive, wrist=wpositive, fatherId=fReference[0]}
  [1265] = {x=-6.277, y=0.000, z=-10.247, rx=-0.000, ry=0.000, rz=-0.000, shoulder=lefty, elbow=epositive, wrist=wpositive, fatherId=fReference[0]}
  [1266] = {x=-6.780, y=0.000, z=-10.256, rx=-0.000, ry=0.000, rz=-0.000, shoulder=lefty, elbow=epositive, wrist=wpositive, fatherId=fReference[0]}
  [1267] = {x=-7.283, y=0.000, z=-10.266, rx=-0.000, ry=0.000, rz=-0.000, shoulder=lefty, elbow=epositive, wrist=wpositive, fatherId=fReference[0]}
  [1268] = {x=-7.786, y=0.000, z=-10.275, rx=-0.000, ry=0.000, rz=-0.000, shoulder=lefty, elbow=epositive, wrist=wpositive, fatherId=fReference[0]}
  [1269] = {x=-8.288, y=0.000, z=-10.285, rx=-0.000, ry=0.000, rz=-0.000, shoulder=lefty, elbow=epositive, wrist=wpositive, fatherId=fReference[0]}
  [1270] = {x=-8.790, y=0.000, z=-10.295, rx=-0.000, ry=0.000, rz=-0.000, shoulder=lefty, elbow=epositive, wrist=wpositive, fatherId=fReference[0]}
  [1271] = {x=-9.292, y=0.000, z=-10.306, rx=-0.000, ry=0.000, rz=-0.000, shoulder=lefty, elbow=epositive, wrist=wpositive, fatherId=fReference[0]}
  [1272] = {x=-9.795, y=0.000, z=-10.316, rx=-0.000, ry=0.000, rz=-0.000, shoulder=lefty, elbow=epositive, wrist=wpositive, fatherId=fReference[0]}
  [1273] = {x=-10.298, y=0.000, z=-10.326, rx=-0.000, ry=0.000, rz=-0.000, shoulder=lefty, elbow=epositive, wrist=wpositive, fatherId=fReference[0]}
  [1274] = {x=-10.801, y=0.000, z=-10.336, rx=-0.000, ry=0.000, rz=-0.000, shoulder=lefty, elbow=epositive, wrist=wpositive, fatherId=fReference[0]}
  [1275] = {x=-11.305, y=0.000, z=-10.346, rx=-0.000, ry=0.000, rz=-0.000, shoulder=lefty, elbow=epositive, wrist=wpositive, fatherId=fReference[0]}
  [1276] = {x=-11.808, y=0.000, z=-10.356, rx=-0.000, ry=0.000, rz=-0.000, shoulder=lefty, elbow=epositive, wrist=wpositive, fatherId=fReference[0]}
  [1277] = {x=-12.311, y=0.000, z=-10.366, rx=-0.000, ry=0.000, rz=-0.000, shoulder=lefty, elbow=epositive, wrist=wpositive, fatherId=fReference[0]}
  [1278] = {x=-12.814, y=0.000, z=-10.376, rx=-0.000, ry=0.000, rz=-0.000, shoulder=lefty, elbow=epositive, wrist=wpositive, fatherId=fReference[0]}
  [1279] = {x=-13.317, y=0.000, z=-10.387, rx=-0.000, ry=0.000, rz=-0.000, shoulder=lefty, elbow=epositive, wrist=wpositive, fatherId=fReference[0]}
  [1280] = {x=-13.821, y=0.000, z=-10.397, rx=-0.000, ry=0.000, rz=-0.000, shoulder=lefty, elbow=epositive, wrist=wpositive, fatherId=fReference[0]}
  [1281] = {x=-14.325, y=0.000, z=-10.408, rx=-0.000, ry=0.000, rz=-0.000, shoulder=lefty, elbow=epositive, wrist=wpositive, fatherId=fReference[0]}
  [1282] = {x=-14.828, y=0.000, z=-10.418, rx=-0.000, ry=0.000, rz=-0.000, shoulder=lefty, elbow=epositive, wrist=wpositive, fatherId=fReference[0]}
  [1283] = {x=-15.331, y=0.000, z=-10.429, rx=-0.000, ry=0.000, rz=-0.000, shoulder=lefty, elbow=epositive, wrist=wpositive, fatherId=fReference[0]}
  [1284] = {x=-15.831, y=0.000, z=-10.440, rx=-0.000, ry=0.000, rz=-0.000, shoulder=lefty, elbow=epositive, wrist=wpositive, fatherId=fReference[0]}
  [1285] = {x=-16.330, y=0.000, z=-10.452, rx=-0.000, ry=0.000, rz=-0.000, shoulder=lefty, elbow=epositive, wrist=wpositive, fatherId=fReference[0]}
  [1286] = {x=-16.827, y=0.000, z=-10.465, rx=-0.000, ry=0.000, rz=-0.000, shoulder=lefty, elbow=epositive, wrist=wpositive, fatherId=fReference[0]}
  [1287] = {x=-17.331, y=0.000, z=-10.478, rx=-0.000, ry=0.000, rz=-0.000, shoulder=lefty, elbow=epositive, wrist=wpositive, fatherId=fReference[0]}
  [1288] = {x=-17.828, y=0.000, z=-10.490, rx=-0.000, ry=0.000, rz=-0.000, shoulder=lefty, elbow=epositive, wrist=wpositive, fatherId=fReference[0]}
  [1289] = {x=-18.316, y=0.000, z=-10.504, rx=-0.000, ry=0.000, rz=-0.000, shoulder=lefty, elbow=epositive, wrist=wpositive, fatherId=fReference[0]}
  [1290] = {x=-18.812, y=0.000, z=-10.518, rx=-0.000, ry=0.000, rz=-0.000, shoulder=lefty, elbow=epositive, wrist=wpositive, fatherId=fReference[0]}
  [1291] = {x=-19.302, y=0.000, z=-10.532, rx=-0.000, ry=0.000, rz=-0.000, shoulder=lefty, elbow=epositive, wrist=wpositive, fatherId=fReference[0]}
  [1292] = {x=-19.798, y=0.000, z=-10.546, rx=-0.000, ry=0.000, rz=-0.000, shoulder=lefty, elbow=epositive, wrist=wpositive, fatherId=fReference[0]}
  [1293] = {x=-20.296, y=0.000, z=-10.560, rx=-0.000, ry=0.000, rz=-0.000, shoulder=lefty, elbow=epositive, wrist=wpositive, fatherId=fReference[0]}
  [1294] = {x=-20.784, y=0.000, z=-10.576, rx=-0.000, ry=0.000, rz=-0.000, shoulder=lefty, elbow=epositive, wrist=wpositive, fatherId=fReference[0]}
  [1295] = {x=-21.284, y=0.000, z=-10.591, rx=-0.000, ry=0.000, rz=-0.000, shoulder=lefty, elbow=epositive, wrist=wpositive, fatherId=fReference[0]}
  [1296] = {x=-21.778, y=0.000, z=-10.606, rx=-0.000, ry=0.000, rz=-0.000, shoulder=lefty, elbow=epositive, wrist=wpositive, fatherId=fReference[0]}
  [1297] = {x=-22.265, y=0.000, z=-10.623, rx=-0.000, ry=0.000, rz=-0.000, shoulder=lefty, elbow=epositive, wrist=wpositive, fatherId=fReference[0]}
  [1298] = {x=-22.761, y=0.000, z=-10.639, rx=-0.000, ry=0.000, rz=-0.000, shoulder=lefty, elbow=epositive, wrist=wpositive, fatherId=fReference[0]}
  [1299] = {x=-23.257, y=0.000, z=-10.657, rx=-0.000, ry=0.000, rz=-0.000, shoulder=lefty, elbow=epositive, wrist=wpositive, fatherId=fReference[0]}
  [1300] = {x=-23.745, y=0.000, z=-10.675, rx=-0.000, ry=0.000, rz=-0.000, shoulder=lefty, elbow=epositive, wrist=wpositive, fatherId=fReference[0]}
  [1301] = {x=-24.242, y=0.000, z=-10.695, rx=-0.000, ry=0.000, rz=-0.000, shoulder=lefty, elbow=epositive, wrist=wpositive, fatherId=fReference[0]}
  [1302] = {x=-24.740, y=0.000, z=-10.714, rx=-0.000, ry=0.000, rz=-0.000, shoulder=lefty, elbow=epositive, wrist=wpositive, fatherId=fReference[0]}
  [1303] = {x=-25.239, y=0.000, z=-10.735, rx=-0.000, ry=0.000, rz=-0.000, shoulder=lefty, elbow=epositive, wrist=wpositive, fatherId=fReference[0]}
  [1304] = {x=-25.739, y=0.000, z=-10.757, rx=-0.000, ry=0.000, rz=-0.000, shoulder=lefty, elbow=epositive, wrist=wpositive, fatherId=fReference[0]}
  [1305] = {x=-26.246, y=0.000, z=-10.782, rx=-0.000, ry=0.000, rz=-0.000, shoulder=lefty, elbow=epositive, wrist=wpositive, fatherId=fReference[0]}
  [1306] = {x=-26.761, y=0.000, z=-10.810, rx=-0.000, ry=0.000, rz=-0.000, shoulder=lefty, elbow=epositive, wrist=wpositive, fatherId=fReference[0]}
  [1307] = {x=-27.280, y=0.000, z=-10.840, rx=-0.000, ry=0.000, rz=-0.000, shoulder=lefty, elbow=epositive, wrist=wpositive, fatherId=fReference[0]}
  [1308] = {x=-27.817, y=0.000, z=-10.873, rx=-0.000, ry=0.000, rz=-0.000, shoulder=lefty, elbow=epositive, wrist=wpositive, fatherId=fReference[0]}
  [1309] = {x=-28.352, y=0.000, z=-10.903, rx=-0.000, ry=0.000, rz=-0.000, shoulder=lefty, elbow=epositive, wrist=wpositive, fatherId=fReference[0]}
  [1310] = {x=-28.904, y=0.000, z=-10.926, rx=-0.000, ry=0.000, rz=-0.000, shoulder=lefty, elbow=epositive, wrist=wpositive, fatherId=fReference[0]}
  [1311] = {x=-28.904, y=0.000, z=289.074, rx=-0.000, ry=0.000, rz=-0.000, shoulder=lefty, elbow=epositive, wrist=wpositive, fatherId=fReference[0]}
  [1312] = {x=-35.000, y=0.000, z=300.000, rx=-0.000, ry=0.000, rz=-0.000, shoulder=lefty, elbow=epositive, wrist=wpositive, fatherId=fReference[0]}
public tool tTool = {x=-0.047, y=0.112, z=264.182, rx=180.000, ry=0.000, rz=-0.000, fatherId=flange[0], ioLink=valve1}
